		IF bSetupModeA THEN
			CASE nSetupModeAStep OF
			0:	(*MM_SetupModeA *)
				IF bMachineFault THEN
					(* Doors closed handled in Faults *)
					bSetupA:=FALSE;
					bACoolantSolenoid := FALSE;
					bSetupModeA:=FALSE;
					nManualModeState:=MM_Nothing;
				(* High Pressure Pump must be running *)
				ELSIF NOT bHighPressureMotorRunning THEN
					bSetupA:=FALSE;
					bACoolantSolenoid := FALSE;
					nManualModeState:=MM_Nothing;
					bSetupModeA:=FALSE;
					nModeError := Er_CoolantOff;
				(* Parts Must be Present *)
				ELSIF NOT(nAEjectorRetractedState=0) OR NOT(nAEjectorAdvancedState=7)
				THEN
					bSetupA:=FALSE;
					bACoolantSolenoid := FALSE;
					nManualModeState:=MM_Nothing;
					bSetupModeA:=FALSE;
					nModeError := Er_SetupError;
					nSetupErrorID:=1;
				(* Parts Must be Clamped *)
				ELSIF NOT(bPS617) THEN
					bSetupA:=FALSE;
					bACoolantSolenoid := FALSE;
					nManualModeState:=MM_Nothing;
					bSetupModeA:=FALSE;
					nModeError := Er_SetupError;
					nSetupErrorID:=2;
				(* UnClamp PS Must be Off *)
				ELSIF bPS616 THEN
					bSetupA:=FALSE;
					bACoolantSolenoid := FALSE;
					nManualModeState:=MM_Nothing;
					bSetupModeA:=FALSE;
					nModeError := Er_SetupError;
					nSetupErrorID:=3;
				(* Exit When Drill Return is Pressed *)
				ELSIF NOT(bPB4ADrillReturn) OR NOT(bPB4BDrillReturn) THEN
					bACoolantSolenoid := FALSE;
					bSetupA:=FALSE;
					bSetupModeA:=FALSE;
					nManualModeState:=MM_Nothing;
				(* If PB is pressed again then move to MMSetup with Spindle *)
				ELSIF fbSetupModeATimer.Q AND bEnterSetupPB_A THEN
					nSetupModeAStep:=1;
					bVFD_ARun:=TRUE;
				(* Turn on the In Setup bit and the solenoid *)
				ELSE
					bACoolantSolenoid := TRUE;
					bSetupA:=TRUE;
				END_IF

			1:	(*	MM_SetupModeAWSpindle		*)
				nVFDControlRPM:=LREAL_TO_UINT(fRPMRequest);
				(* The Setup can be canceled by Drill Retrun of Fault Reset *)
				IF bMachineFault OR NOT(bPB4ADrillReturn) OR NOT(bPB4BDrillReturn) OR bFaultResetPB THEN
					bACoolantSolenoid :=FALSE;
					bVFD_ARun:=FALSE;
					bSetupA:=FALSE;
					bSetupModeA:=FALSE;
					nSetupModeAStep:=0;
					nManualModeState:=MM_Nothing;
				END_IF
			END_CASE	(* nSetupModeAStep *)
		END_IF (*bSetupmodeA *)

		(* MM_SetupModeB*)
		IF bSetupModeB THEN
			CASE nSetupModeBStep OF
			0:	(*MM_SetupModeB *)
				IF bMachineFault THEN
					(* Doors closed handled in Faults *)
					bSetupB:=FALSE;
					bBCoolantSolenoid := FALSE;
					bSetupModeB:=FALSE;
					nManualModeState:=MM_Nothing;
				(* High Pressure Pump must be running *)
				ELSIF NOT bHighPressureMotorRunning THEN
					bSetupB:=FALSE;
					bBCoolantSolenoid := FALSE;
					nManualModeState:=MM_Nothing;
					bSetupModeB:=FALSE;
					nModeError := Er_CoolantOff;
				(* Parts Must be Present *)
				ELSIF NOT(nBEjectorRetractedState=0) OR NOT(nBEjectorAdvancedState=7)
				THEN
					bSetupB:=FALSE;
					bBCoolantSolenoid := FALSE;
					nManualModeState:=MM_Nothing;
					bSetupModeB:=FALSE;
					nModeError := Er_SetupError;
					nSetupErrorID:=1;
				(* Parts Must be Clamped *)
				ELSIF NOT(bPS727) THEN
					bSetupB:=FALSE;
					bBCoolantSolenoid := FALSE;
					nManualModeState:=MM_Nothing;
					bSetupModeB:=FALSE;
					nModeError := Er_SetupError;
					nSetupErrorID:=2;
				(* Unclamped PS Off*)
				ELSIF bPS726 THEN
					bSetupB:=FALSE;
					bBCoolantSolenoid := FALSE;
					nManualModeState:=MM_Nothing;
					bSetupModeB:=FALSE;
					nModeError := Er_SetupError;
					nSetupErrorID:=3;
				(* Exit When Drill Return is Pressed *)
				ELSIF NOT(bPB4ADrillReturn) OR NOT(bPB4BDrillReturn) THEN
					bBCoolantSolenoid := FALSE;
					bSetupB:=FALSE;
					bSetupModeB:=FALSE;
					nManualModeState:=MM_Nothing;
				(* If PB is pressed again then move to MMSetup with Spindle *)
				ELSIF fbSetupModeBTimer.Q AND bEnterSetupPB_B THEN
					nSetupModeBStep:=1;
					bVFD_BRun:=TRUE;
				(* Turn on the In Setup bit and the solenoid *)
				ELSE
					bBCoolantSolenoid := TRUE;
					bSetupB:=TRUE;
				END_IF

			1:	(*MM_SetupModeBWSpindle*)
				nVFDControlRPM:=LREAL_TO_UINT(fRPMRequest);
				(* The Setup can be canceled by Drill Retrun of Fault Reset *)
				IF bMachineFault OR NOT(bPB4ADrillReturn) OR NOT(bPB4BDrillReturn) OR bFaultResetPB THEN
					bBCoolantSolenoid :=FALSE;
					bVFD_BRun:=FALSE;
					bSetupB:=FALSE;
					bSetupModeB:=FALSE;
					nSetupModeBStep:=0;
					nManualModeState:=MM_Nothing;
				END_IF
			END_CASE	(* nSetupModeAStep *)
		END_IF (*bSetupmodeB *)

		MM_SetZAZero:
			IF bMachineFault THEN
				bZAAxisSetZero := FALSE;
				nManualModeState:=MM_Nothing;
			ELSIF fbZAAxisSetZero.Error THEN
				nModeError := Er_ZAHomeError;
				bZAAxisSetZero := FALSE;
				nManualModeState:=MM_Nothing;
			ELSIF fbZAAxisSetZero.Done THEN
				bZAAxisSetZero := FALSE;
				nManualModeState:=MM_Nothing;
			ELSE
				bZAAxisSetZero := TRUE;
			END_IF

		MM_SetZBZero:
			IF bMachineFault THEN
				bZBAxisSetZero := FALSE;
				nManualModeState:=MM_Nothing;
			ELSIF fbZBAxisSetZero.Error THEN
				nModeError := Er_ZBHomeError;
				bZBAxisSetZero := FALSE;
				nManualModeState:=MM_Nothing;
			ELSIF fbZBAxisSetZero.Done THEN
				bZBAxisSetZero := FALSE;
				nManualModeState:=MM_Nothing;
			ELSE
				bZBAxisSetZero := TRUE;
			END_IF

		MM_MoveZAToZero:
			IF bMachineFault THEN
				bZAAxisMove := FALSE;
				nManualModeState:=MM_Nothing;
			ELSIF fbZAAxisMove.Error THEN
				nModeError := Er_ZAMoveError;
				bZAAxisMove := FALSE;
				nManualModeState:=MM_Nothing;
			ELSIF fbZAAxisMove.Done THEN
				bZAAxisMove := FALSE;
				nManualModeState:=MM_Nothing;
			ELSE
				bZAAxisMove := TRUE;
				fZAMovePosition := 0.0;
				fZAMoveVelocity := 25.0;
			END_IF

		MM_MoveZBToZero:
			IF bMachineFault THEN
				bZBAxisMove := FALSE;
				nManualModeState:=MM_Nothing;
			ELSIF fbZBAxisMove.Error THEN
				nModeError := Er_ZBMoveError;
				bZBAxisMove := FALSE;
				nManualModeState:=MM_Nothing;
			ELSIF fbZBAxisMove.Done THEN
				bZBAxisMove := FALSE;
				nManualModeState:=MM_Nothing;
			ELSE
				bZBAxisMove := TRUE;
				fZBMovePosition := 0.0;
				fZBMoveVelocity := 25.0;
			END_IF

		MM_CoolantOn:
			(* Make sure the Clean tank level has been on for 2 seconds so that we
				don't draw the level down to quickly when we start the High Pressure Pump *)
			fbCleanTankLevelDelay(IN:=bCleanTankLevel, PT:=t#2s);
			(* If the Coolant Stop PB is pressed while in startup *)
			IF bCoolantStopPB THEN
				nManualModeState:=MM_CoolantOff;
			END_IF

			IF bMachineFault THEN
				bHPCoolantStart_A :=FALSE;
				bHPCoolantStart_B :=FALSE;
				bTransferPumpMotorControl:=FALSE;
				bHighPressureMotorControl:=FALSE;
				nManualModeState:=MM_Nothing;
			(* S1: Start the transfer pump and Turn on the Soft Start Solenoid Valves *)
			ELSIF NOT(fbSoftStartTimer.Q) AND NOT(fbSoftStartTimer2.Q) THEN
				bHPCoolantStart_A :=TRUE;
				bHPCoolantStart_B :=TRUE;
				bTransferPumpMotorControl:=TRUE;
			(* S2: After 5 seconds turn on high pressure Motor *)
			(* Note: We can stay here until we get a fault such as Low Tank Level *)
			ELSIF fbSoftStartTimer.Q AND NOT(fbSoftStartTimer2.Q) AND fbCleanTankLevelDelay.Q
				AND NOT(bCoolantTempWarning) AND bCoolantTankOverflow
			THEN
				bHighPressureMotorControl:=TRUE;
			(* S3: After 5 more seconds Turn off the Soft Start Solenoids *)
			ELSIF fbSoftStartTimer2.Q THEN
				bHPCoolantStart_A :=FALSE;
				bHPCoolantStart_B :=FALSE;
				bChipConveyorMotorControl:=TRUE;
				nManualModeState:=MM_Nothing;
			END_IF

		MM_CoolantOff:
			(*	Turn off High Pressure Motor *)
			bHighPressureMotorControl:=FALSE;
			(* Do not shut off the transfer pump until the coolant temp is below the warning *)
			IF bCoolantTempWarning OR bCoolantTempFault THEN
				bChipConveyorMotorControl:=FALSE;
				nManualModeState:=MM_Nothing;
			ELSIF NOT(bHighPressureMotorOn) THEN
				(*	Turn off Transfer Pump *)
				bTransferPumpMotorControl:=FALSE;
				(*	Done *)
				IF NOT(bTransferPumpOn) THEN
					bChipConveyorMotorControl:=FALSE;
					nManualModeState:=MM_Nothing;
				END_IF
			END_IF

		MM_HomeAutomation:
			IF bMachineFault THEN
				nHomeAutomationStep:=0;
				bWAAxisHome:=FALSE;
				bWBAxisHome:=FALSE;
				bUAxisHome:=FALSE;
				(* Trigger MCStop of Axis.  The bits are turned false when done in respective control *)
				bWAStop:=TRUE;
				bWAStop:=TRUE;
				bUStop:=TRUE;
			ELSE
				CASE nHomeAutomationStep OF
				0: (* Trigger Home of WA and WB Axis *)
					IF bSideAEnabled THEN
						bWAAxisHome:=TRUE;	(* Turned off in P_Tailstock Control PRG *)
					END_IF
					IF bSideBEnabled THEN
						bWBAxisHome:=TRUE;	(* Turned off in P_Tailstock Control PRG *)
					END_IF
					nHomeAutomationStep:=nHomeAutomationStep+1;
	
				1: (* After 1 second then start Homing the U Axis, This assures enough clearance *)
					fbHomeTimer(IN:=TRUE, PT:=t#2s);
					IF fbHomeTimer.Q THEN
						fbHomeTimer(IN:=FALSE);
						(* If an error occurs in either of the Axis we want leave the homing operation *)
						IF fbWAAxisHome.Error OR fbHomeWB.Error THEN
							nHomeAutomationStep:=0;
							nManualModeState:=MM_Nothing;
						(* No Errors Move On *)
						ELSE
							bUAxisHome:=TRUE;
							nHomeAutomationStep:=nHomeAutomationStep+1;
						END_IF
					END_IF
	
				2: (* Check for Done bits of the three Axis *)
					fbHomeTimer(IN:=TRUE, PT:=t#90s);
					(* When All Axis are Homed we return *)
					IF (stWAAxis.NcToPlc.StateDWord.1 AND stWBAxis.NcToPlc.StateDWord.1 AND stUAxis.NcToPlc.StateDWord.1) OR
						(* or if an Error occurs *)
						 fbWAAxisHome.Error OR fbHomeWB.Error OR fbTransferAxisHome.Error OR
						(* or if Homing takes too long *)
						fbHomeTimer.Q
					THEN
						fbHomeTimer(IN:=FALSE);
						nHomeAutomationStep:=0;
						nManualModeState:=MM_Nothing;
						IF fbHomeTimer.Q THEN
							nModeError:=Er_HomeTimeout;
						END_IF
					END_IF

				END_CASE	(* nHomeAutomationStep *)
			END_IF	(* Fault check of MM_HomeAutomation *)

		END_CASE	(* Manual Mode State *)

	(*********		AUTOMATIC MODE 		***********)
	ELSE
		CASE nAutoModeState OF
		AM_NotInCycle:
			(* If we have a fault we Exit Auto Mode *)
			IF bMachineFault THEN
				bMachineMode:=FALSE;
			(* We disable cycle start when we have warings *)
			ELSIF bCycleStartControlEnable AND NOT(bMachineWarning)  THEN
				(* Doors will fault if not closed in cycle *)
				nAutoModeState:=AM_RetractZAxis;
			END_IF

		AM_RetractZAxis:
			IF bMachineFault THEN
				bZAAxisMove:= FALSE;
				bZBAxisMove:= FALSE;
				bZAStop := TRUE;
				bZBStop := TRUE;
				nAutoModeState:=AM_NotInCycle;
			ELSE
				(* Move Z axis to Drill Tip Offset Position *)
				IF bSideAEnabled THEN
					bZAAxisMove:= TRUE;
					fZAMovePosition := fDrillTipOffset;
					fZAMoveVelocity := 25;
				END_IF
				IF bSideBEnabled THEN
					bZBAxisMove:= TRUE;
					fZBMovePosition := fDrillTipOffset;
					fZBMoveVelocity := 25;
				END_IF
				(* Stop Axis and Fault if Move Error *)
				IF (bSideAEnabled AND fbZAAxisMove.Error) THEN
					bZAAxisMove:= FALSE;
					nModeError := Er_ZAHomeError;
					bZAStop:=TRUE;	(* Issue a Stop Axis *)
					bZBAxisMove:= FALSE;
					bMachineMode:=FALSE;	(* Go to Manual Mode *)
				ELSIF (bSideBEnabled AND fbZBAxisMove.Error) THEN
					bZBAxisMove:= FALSE;
					nModeError := Er_ZAHomeError;
					bZBStop:=TRUE;	(* Issue a Stop Axis *)
					bZAAxisMove:= FALSE;
					bMachineMode:=FALSE;	(* Go to Manual Mode *)
				(* If Move Done we Go Into Cycle *)
				ELSIF (NOT(bSideAEnabled) OR fbZAAxisMove.Done) AND
					(NOT(bSideBEnabled) OR fbZBAxisMove.Done) THEN
					bZAAxisMove:= FALSE;
					bZBAxisMove:= FALSE;
					nAutoModeState:=AM_InCycle;
				END_IF
			END_IF

		AM_InCycle:
			(* These Things Happen While In Cycle *)
			fbCoolantTimer(IN:=bCoolantTimer , PT:=tCoolantTime);
			fbCycleTimer(IN:=bCycleTimer , PT:=t#10h);
			(* If the Load confirm PB has been pressed and the parts are there,  then Set a bit for Load Confirm *)
			IF ( sLoadSideSet = 'A' AND bPB1AConfirm AND
				(NOT(bSideAEnabled) OR bProx410 AND bProx411 AND bProx412) AND
				(NOT(bSideBEnabled) OR bProx413 AND bProx414 AND bProx415) ) OR
				(sLoadSideSet ='B' AND bPB1BConfirm AND
				( NOT(bSideAEnabled) OR bProx510 AND bProx511 AND bProx512) AND
				(NOT(bSideBEnabled) OR bProx513 AND bProx514 AND bProx515) )
			THEN
				bLoadPartsConfirmed:= TRUE;	(* Turned Off in Transfer Control *)
			(* Else Set a Warning that Parts are Missing when the PB pressed
				We want to ignore the PB if we have already confirmed parts loaded *)
			ELSIF NOT bLoadPartsConfirmed AND
				( sLoadSideSet = 'A' AND fbPB1AConfirmRTrig.Q) OR
				(sLoadSideSet ='B' AND fbPB1BConfirmRTrig.Q)
			THEN
				nModeError:=Er_LoadPartMissing;
			END_IF
			(* If the Unloadoad confirm PB's have been pressed and there are no parts,  then Set a bit for Unload Confirm *)
			IF (sLoadSideSet = 'B' AND fbPB1AConfirmRTrig.Q AND
				NOT(bProx410 OR bProx411 OR bProx412 OR bProx413 OR bProx414 OR bProx415) ) OR
				(sLoadSideSet ='A' AND fbPB1BConfirmRTrig.Q AND
				NOT(bProx510 OR bProx511 OR bProx512 OR bProx513 OR bProx514 OR bProx515) )
			THEN
				bUnloadPartsConfirmed:= TRUE;
			(* Else set a Warning that Parts are present *)
			ELSIF (sLoadSideSet = 'B' AND fbPB1AConfirmRTrig.Q) OR (sLoadSideSet ='A' AND fbPB1BConfirmRTrig.Q) THEN
				nModeError:=Er_UnloadPartPresent;
			END_IF

			(*	Implement Auto Cycle Stuff Here *)
			CASE nAutoCycleStep OF
			AC_Init:
				bCycleStartControlHold:=FALSE;
				bCycleStartControlReset:=FALSE;
				bCycleTimer:=FALSE;
				(* Check Faults *)
				IF bMachineFault THEN (* Added V1.5 *)
					bInCycle:=FALSE;
					bMachineMode:=FALSE;
					bCycleStartControlReset:=TRUE;
					nAutoModeState:=AM_NotInCycle;
				ELSIF bLoadPartsConfirmed THEN
					nDrillStep := 0;
					bInCycle:=TRUE;
					nAutoCycleStep:=AC_TransferParts;
				END_IF

			AC_TransferParts:
				(* When Cycle Counter Reached and not Cell Runout we Fault *)
				IF (nCyclesComplete >= nMaxCycles) AND NOT bCellRunoutRequest THEN
					nModeError:= Er_MaxCyclesReached;
					nAutoCycleStep:=AC_Init;
					nAutoModeState:=AM_NotInCycle;
					bMachineMode:=FALSE;
					bCycleStartControlReset:=TRUE;
					bCycleStartControlHold:=FALSE;
					bCycleWatchdogTimer := FALSE;
					bInCycle:=FALSE;
					bCycleTimer:=FALSE;
					bDisplayUnloadConf := FALSE;
				ELSE
					bCycleTimer:=TRUE;
					IF bMachineFault OR fbCycleWatchdogTimer.Q THEN
						nAutoCycleStep:=AC_Init;
						bInCycle:=FALSE;
						bMachineMode:=FALSE;
						bCycleStartControlReset:=TRUE;
						bCycleStartControlHold:=FALSE;
						bCycleWatchdogTimer := FALSE;
						bCycleTimer:=FALSE;
						bDisplayUnloadConf := FALSE;
						bAutoTransferPartsToDrill:=FALSE;
						nAutoModeState:=AM_NotInCycle;
					(* At Unload Position and UP, So Go to Clamp *)
					ELSIF bTransferAtUnloadIndicator AND
						bProx516 AND NOT(bProx517)
					THEN
						bCycleWatchdogTimer := FALSE;
						IF nCellRunoutCounter=1 AND bCellRunoutRequest THEN
							nAutoCycleStep:=AC_CellRunoutFinish;
						ELSE
							nAutoCycleStep:=AC_Clamp;
						END_IF
					(* Trigger Transfer Move *)
					ELSIF NOT bAutoTransferPartsToDrill  AND bUnloadPartsConfirmed THEN
						bDisplayUnloadConf := FALSE;
						bAutoTransferPartsToDrill:=TRUE;
						bCycleWatchdogTimer := TRUE;
						tCycleWatchdogTime := t#120s;
					(* Display Waiting on Unload Confirm Button *)
					ELSIF NOT bUnloadPartsConfirmed THEN
						bDisplayUnloadConf := TRUE;
					END_IF
				END_IF (* Max Cycles Check *)

			AC_Clamp:
				IF bMachineFault (* OR fbCycleWatchdogTimer.Q *) THEN
					nAutoCycleStep:=AC_Init;
					bInCycle:=FALSE;
					bMachineMode:=FALSE;
					bCycleStartControlReset:=TRUE;
					bCycleStartControlHold:=FALSE;
					bCycleTimer:=FALSE;
					bCycleWatchdogTimer := FALSE;
					bAutoClampAStart:=FALSE;
					bAutoClampBStart:=FALSE;
					nAutoModeState:=AM_NotInCycle;
				(* Done Clamping so Go To Coolant On *)
				ELSIF(bAutoClampADone OR NOT(bSideAEnabled)) AND
						(bAutoClampBDone OR NOT(bSideBEnabled)) THEN
					bAutoTransferDownAndLoad := TRUE;
					bCycleWatchdogTimer := FALSE;
					nAutoCycleStep:=AC_CoolantOn;
				(* Trigger Clamping *)
				ELSE
					bCycleWatchdogTimer := TRUE;
					tCycleWatchdogTime := t#30s;
					IF bSideAEnabled THEN
						bAutoClampAStart:=TRUE;
					END_IF
					IF bSideBEnabled THEN
						bAutoClampBStart:=TRUE;
					END_IF
				END_IF

			AC_CoolantOn:
				IF bMachineFault OR fbCycleWatchdogTimer.Q THEN
					nAutoCycleStep:=AC_Init;
					bInCycle:=FALSE;
					bMachineMode:=FALSE;
					bCycleStartControlReset:=TRUE;
					bCycleStartControlHold:=FALSE;
					bCycleTimer:=FALSE;
					bCycleWatchdogTimer := FALSE;
					bAutoClampAStart:=FALSE;
					bAutoClampBStart:=FALSE;
					bACoolantSolenoid:=FALSE;
					bBCoolantSolenoid:=FALSE;
					bAutoTransferDownAndLoad := FALSE;
					IF fbCycleWatchdogTimer.Q THEN
						nModeError:=Er_AMCoolantTimeout;
					END_IF
					nAutoModeState:=AM_NotInCycle;
				(* S2: When Pressure Switch On Delay then Turn Spindles On *)
				ELSIF (fbPS1DelayTON.Q OR NOT(bSideAEnabled)) AND
						(fbPS2DelayTON.Q OR NOT(bSideBEnabled)) THEN
					bCycleWatchdogTimer := FALSE;
					nAutoCycleStep:=AC_SpindleOn;
				(* S1: Turn on the Coolant and start the watchdog Timer
					Set the PS delay timer *)
				ELSE
					IF bSideAEnabled THEN
						bACoolantSolenoid:=TRUE;
					END_IF
					IF bSideBEnabled THEN
						bBCoolantSolenoid:=TRUE;
					END_IF
					tCoolantTime:= t#1.5s;
					bCycleWatchdogTimer := TRUE;
					tCycleWatchdogTime := t#15s;
				END_IF

			AC_SpindleOn:
				nVFDControlRPM:=LREAL_TO_UINT(fRPMRequest);
				IF bMachineFault OR fbCycleWatchdogTimer.Q THEN
					nAutoCycleStep:=AC_Init;
					bInCycle:=FALSE;
					bMachineMode:=FALSE;
					bCycleStartControlReset:=TRUE;
					bCycleStartControlHold:=FALSE;
					bCycleTimer:=FALSE;
					bCycleWatchdogTimer := FALSE;
					bAutoClampAStart:=FALSE;
					bAutoClampBStart:=FALSE;
					bACoolantSolenoid:=FALSE;
					bBCoolantSolenoid:=FALSE;
					bVFD_ARun:=FALSE;
					bVFD_BRun:=FALSE;
					bAutoTransferDownAndLoad := FALSE;
					IF fbCycleWatchdogTimer.Q THEN
						nModeError:=Er_VFDUpToSpeedTimeout;
					END_IF
					nAutoModeState:=AM_NotInCycle;
				(* S2: Once up to Speed then Drill *)
				ELSIF (fbUpToSpeedATON.Q OR NOT(bSideAEnabled)) AND
						(fbUpToSpeedBTON.Q OR NOT(bSideBEnabled)) THEN
					bCycleWatchdogTimer := FALSE;
					nAutoCycleStep:=AC_Drill;
				(* S1: Turn on Spindles *)
				ELSE
					IF bSideAEnabled THEN
						bVFD_ARun := TRUE;
					END_IF
					IF bSideBEnabled THEN
						bVFD_BRun := TRUE;
					END_IF
					tCycleDelayTime := t#250ms;
				END_IF

			AC_Drill:
				(* Safety interlock: while drilling, keep transfer commands disabled so the part cannot move with drills engaged. *)
				bAutoTransferPartsToDrill:=FALSE;
				bAutoTransferDownAndLoad:=FALSE;
				IF bMachineFault  AND
					(*Faults Array 4 are ones that should not stop the drill cycle *)
					NOT( nActiveFaults[4]>0
						AND nActiveFaults[1]=0
						AND nActiveFaults[2]=0
						AND nActiveFaults[3]=0)
				THEN
					nAutoCycleStep:=AC_DrillReturn;
					nDrillStep := 0;
					bInCycle:=FALSE;
					bCycleStartControlReset:=TRUE;
					bCycleStartControlHold:=FALSE;
					bCycleTimer:=FALSE;
					bCycleWatchdogTimer := FALSE;
					bAutoClampAStart:=FALSE;
					bAutoClampBStart:=FALSE;
					bACoolantSolenoid:=FALSE;
					bBCoolantSolenoid:=FALSE;
					bZAAxisMove:=FALSE;
					bZBAxisMove:=FALSE;
					bZAStop := TRUE;
					bZBStop := TRUE;
					bVFD_ARun:=FALSE;
					bVFD_BRun:=FALSE;
					bDwellTime:= FALSE;
					bAutoTransferDownAndLoad := FALSE;
				ELSE
					(* S1: Move to Strart Depth at Startfeed *)
					(* S2: Wait for Move Done bit *)
					(* S3: Move to Finish Depth at Finish Feed *)
					(* S4: Wait for Move Done bit *)
					(* S5: If Dead Spindle Retract Then-Turn off Spindles *)
					(* T5: VFD's at Zero Speed *)
					(* S6: If Not Dead Spindle Retract then use Dwell Timer *)
					CASE nDrillStep OF
					0: (* S1: Set Execute for Z Axis *)
						IF bSideAEnabled THEN
							bZAAxisMove:=TRUE;
							fZAMovePosition:= fStartDepth;
							fZAMoveVelocity:= fStartFeed/60;
						END_IF
						IF bSideBEnabled THEN
							bZBAxisMove:=TRUE;
							fZBMovePosition:= fStartDepth;
							fZBMoveVelocity:= fStartFeed/60;
						END_IF
						(* T1: Wait for Busy bit *)
						IF (fbZAAxisMove.Busy OR NOT(bSideAEnabled)) AND
							(fbZBAxisMove.Busy OR NOT(bSideBEnabled)) THEN
							nDrillStep:=nDrillStep+1;
						END_IF

					1:(* S2: Wait for Move Start Depth Done bit *)
						IF (fbZAAxisMove.Done OR NOT(bSideAEnabled)) AND
							(fbZBAxisMove.Done OR NOT(bSideBEnabled)) THEN
							bZAAxisMove:=FALSE;
							bZBAxisMove:=FALSE;
							nDrillStep:=nDrillStep+1;
						END_IF

					2: (* S3: Move to Finish Depth at Finish Feed *)
						IF bSideAEnabled THEN
							bZAAxisMove:=TRUE;
							fZAMovePosition:= fFinishDepth;
							fZAMoveVelocity:= fFinishFeed/60;
						END_IF
						IF bSideBEnabled THEN
							bZBAxisMove:=TRUE;
							fZBMovePosition:= fFinishDepth;
							fZBMoveVelocity:= fFinishFeed/60;
						END_IF
						(* T1: Wait for Busy bit *)
						IF (fbZAAxisMove.Busy OR NOT(bSideAEnabled)) AND
							(fbZBAxisMove.Busy OR NOT(bSideBEnabled)) THEN
							nDrillStep:=nDrillStep+1;
						END_IF

					3: (* S4: Wait for Move Done bit *)
						IF (fbZAAxisMove.Done OR NOT(bSideAEnabled)) AND
							(fbZBAxisMove.Done OR NOT(bSideBEnabled)) THEN
							bZAAxisMove:=FALSE;
							bZBAxisMove:=FALSE;
							nDrillStep:=nDrillStep+1;
						END_IF

					4: (* If Dead Spindle Retract then go to Step 5, Else Step 6 *)
						IF bSpindleRetractMode THEN
							nDrillStep:=nDrillStep+1;
						ELSE
							nDrillStep:=6;
						END_IF

					5: (* S5: Turn off Spindles *)
						(* Turn off the VFD Run singnals *)
						bVFD_ARun:=FALSE;
						bVFD_BRun:=FALSE;
						tCycleWatchdogTime := t#5s;
						bCycleWatchdogTimer:=TRUE;
						IF (NOT(bSideAEnabled) OR (stVFD_A1DriveInfo.nActualSpeed < 5) OR
							(stVFD_A2DriveInfo.nActualSpeed < 5) OR (stVFD_A3DriveInfo.nActualSpeed < 5) )
							AND (NOT(bSideBEnabled) OR  (stVFD_A1DriveInfo.nActualSpeed < 5) OR
							(stVFD_A2DriveInfo.nActualSpeed < 5) OR (stVFD_A3DriveInfo.nActualSpeed < 5) )
						THEN
							bCycleWatchdogTimer := FALSE;
							nDrillStep:=0;
							nAutoCycleStep:=AC_Retract;
						(* If This took too long then jump to next step *)
						ELSIF fbCycleWatchdogTimer.Q THEN
							bCycleWatchdogTimer := FALSE;
							nDrillStep:=0;
							nAutoCycleStep:=AC_Retract;
						END_IF

					6: (* S6: Dwell Timer *)
						IF fDwellTime > 0.0 THEN
							bDwellTime:= TRUE;
							fbDwellTimeTON(IN:=bDwellTime, PT:=LREAL_TO_TIME(fDwellTime) );
							IF fbDwellTimeTON.Q THEN
								bDwellTime:= FALSE;
								nDrillStep:=0;
								nAutoCycleStep:=AC_Retract;
							END_IF
						ELSE (* No Dwell Time *)
							nDrillStep:=0;
							nAutoCycleStep:=AC_Retract;
						END_IF

					END_CASE
				END_IF

			AC_DrillReturn:
				(* Keep transfer disabled until Z axes have returned to drill tip offset. *)
				bAutoTransferPartsToDrill:=FALSE;
				bAutoTransferDownAndLoad:=FALSE;
				CASE nDrillReturnCount OF
				0: (* Wait for the Stop to finish and Move to Drill Tip Offset *)
					IF NOT bZAStop AND NOT bZBStop THEN
						bZAAxisMove:=TRUE;
						bZBAxisMove:=TRUE;
						fZAMovePosition:=fDrillTipOffset;
						fZBMovePosition:=fDrillTipOffset;
						fZAMoveVelocity:=50;
						fZBMoveVelocity:=50;
						nDrillReturnCount:=nDrillReturnCount+1;
					END_IF

				1: (* Wait for move to be done *)
					IF fbZAAxisMove.Done AND fbZBAxisMove.Done THEN
						bZAAxisMove:=FALSE;
						bZBAxisMove:=FALSE;
						bMachineMode:=FALSE;
						nAutoModeState:=AM_NotInCycle;
						nDrillReturnCount:=0;
					END_IF
				END_CASE


			AC_Retract:
				(* Keep transfer disabled until drills are fully retracted and spindle/coolant shutdown is complete. *)
				bAutoTransferPartsToDrill:=FALSE;
				bAutoTransferDownAndLoad:=FALSE;
				IF bMachineFault  AND
					(*Faults Array 4 are ones that should not stop the drill cycle *)
					NOT( (nActiveFaults[4]>0)
						AND nActiveFaults[1]=0
						AND nActiveFaults[2]=0
						AND nActiveFaults[3]=0)
				THEN
					nAutoCycleStep:=AC_Init;
					nDrillStep := 0;
					bInCycle:=FALSE;
					bMachineMode:=FALSE;
					bCycleStartControlReset:=TRUE;
					bCycleStartControlHold:=FALSE;
					bCycleTimer:=FALSE;
					bCycleWatchdogTimer := FALSE;
					bAutoClampAStart:=FALSE;
					bAutoClampBStart:=FALSE;
					bACoolantSolenoid:=FALSE;
					bBCoolantSolenoid:=FALSE;
					bZAAxisMove:=FALSE;
					bZBAxisMove:=FALSE;
					bZAStop := TRUE;
					bZBStop := TRUE;
					bVFD_ARun:=FALSE;
					bVFD_BRun:=FALSE;
					bAutoTransferDownAndLoad := FALSE;
					nAutoModeState:=AM_NotInCycle;
				(* T1: Move Done Bit *)
				ELSIF (fbZAAxisMove.Done OR NOT(bSideAEnabled)) AND
						(fbZBAxisMove.Done OR NOT(bSideBEnabled)) THEN
					bZAAxisMove:=FALSE;
					bZBAxisMove:=FALSE;
					nAutoCycleStep:=AC_SpindleOff;
				(* S1: Move to Start Position *)
				ELSE
					IF bSideAEnabled THEN
						bZAAxisMove:=TRUE;
						fZAMovePosition:= (0.0 + fDrillTipOffset);
						fZAMoveVelocity:= fRetractRate/60;
					END_IF
					IF bSideBEnabled THEN
						bZBAxisMove:=TRUE;
						fZBMovePosition:= (0.0 + fDrillTipOffset);
						fZBMoveVelocity:= fRetractRate/60;
					END_IF
				END_IF

			AC_SpindleOff:
				(* Turn off the VFD Run singnals *)
				bVFD_ARun:=FALSE;
				bVFD_BRun:=FALSE;
				nAutoCycleStep:=AC_CoolantOff;

			AC_CoolantOff:
				(* Turn off the Coolant Valves *)
				bACoolantSolenoid:=FALSE;
				bBCoolantSolenoid:=FALSE;
				(* Add a time delay so we don't squirt coolant before Unclamping *)
				bCoolantTimer:=TRUE;
				tCoolantTime:=t#250ms;
				IF ( bMachineFault  AND
					(*Faults Array 4 are ones that should not stop the drill cycle *)
					NOT( (nActiveFaults[4]>0)
						AND nActiveFaults[1]=0
						AND nActiveFaults[2]=0
						AND nActiveFaults[3]=0) )
					OR fbCycleWatchdogTimer.Q
				THEN
					nAutoCycleStep:=AC_Init;
					bInCycle:=FALSE;
					bMachineMode:=FALSE;
					bCoolantTimer:=FALSE;
					bCycleStartControlReset:=TRUE;
					bCycleStartControlHold:=FALSE;
					bCycleTimer:=FALSE;
					bCycleWatchdogTimer := FALSE;
					bAutoClampAStart:=FALSE;
					bAutoClampBStart:=FALSE;
					bAutoTransferDownAndLoad := FALSE;
					IF fbCycleWatchdogTimer.Q THEN
						nModeError:=Er_MMCoolantValveStopTimeout;
					END_IF
					nAutoModeState:=AM_NotInCycle;
				ELSIF NOT(bACoolantPressure) AND NOT(bBCoolantPressure) THEN
					bCycleWatchdogTimer := FALSE;
					bCoolantTimer:=FALSE;
					nCyclesComplete:=nCyclesComplete+1;
					IF bSideAEnabled THEN
						nPartsCompleteTotal:=nPartsCompleteTotal+3;
						nPartsCompleteA1:=nPartsCompleteA1+1;
						nPartsCompleteA2:=nPartsCompleteA2+1;
						nPartsCompleteA3:=nPartsCompleteA3+1;
					END_IF
					IF bSideBEnabled THEN
						nPartsCompleteTotal:=nPartsCompleteTotal+3;
						nPartsCompleteB1:=nPartsCompleteB1+1;
						nPartsCompleteB2:=nPartsCompleteB2+1;
						nPartsCompleteB3:=nPartsCompleteB3+1;
					END_IF
					nAutoCycleStep:=AC_Unclamp;
				ELSE
					bCycleWatchdogTimer := TRUE;
					tCycleWatchdogTime := t#10s;
				END_IF

			AC_Unclamp:
				(* Turn off the Clamp Starts *)
				bAutoClampAStart:=FALSE;
				bAutoClampBStart:=FALSE;
				IF ( bMachineFault  AND
					(*Faults Array 4 are ones that should not stop the drill cycle *)
					NOT( (nActiveFaults[4]>0)
						AND nActiveFaults[1]=0
						AND nActiveFaults[2]=0
						AND nActiveFaults[3]=0) )
					OR fbCycleWatchdogTimer.Q
				THEN
					nAutoCycleStep:=AC_Init;
					bInCycle:=FALSE;
					bMachineMode:=FALSE;
					bCycleStartControlReset:=TRUE;
					bCycleStartControlHold:=FALSE;
					bCycleTimer:=FALSE;
					bCycleWatchdogTimer := FALSE;
					bAutoTransferDownAndLoad := FALSE;
					bAutoUpDelayWhileUnclamp := FALSE;
					bAutoUnclampAStart:=FALSE;
					bAutoUnclampBStart:=FALSE;
					nAC_UnclampStep:=0;
					IF fbCycleWatchdogTimer.Q THEN
						nModeError:=Er_AMUnclampTimeout;
					END_IF
					nAutoModeState:=AM_NotInCycle;
				END_IF

				CASE nAC_UnclampStep OF
				0: (* Wait for Transfer to beAt Load Station and Up *)
					IF bTransferAtLoadIndicator AND
						fbProx516TON.Q AND NOT(bProx517)
					THEN
						nAC_UnclampStep := nAC_UnclampStep + 1;
					END_IF

				1: (* Once Delay timer done we can start the Unclamp process *)
					(* Watchdog happens in FB, so we need to make this one longer -
						not necessary, but did not want to remove without parts to run. *)
					bCycleWatchdogTimer := TRUE;
					tCycleWatchdogTime := t#15s;
					(* Unclamp the sides that are enabled *)
					IF bSideAEnabled THEN
						bAutoUnclampAStart:=TRUE;
					END_IF
					IF bSideBEnabled THEN
						bAutoUnclampBStart:=TRUE;
					END_IF
					bUnclampDelayTimer := FALSE;
					nAC_UnclampStep := nAC_UnclampStep + 1;

				2: (* Wait for Unload to be done on the sides that are enabled *)
					(* Unclamp Done, Trigger Transfer *)
					IF (NOT(bSideAEnabled) OR bAutoUnclampADone) AND
							(NOT(bSideBEnabled) OR bAutoUnclampBDone) THEN
						bAutoUnclampAStart:=FALSE;
						bAutoUnclampBStart:=FALSE;
						bCycleWatchdogTimer := FALSE;
						bAutoTransferDownAndLoad := FALSE;
						nAC_UnclampStep := 0;
						nAutoCycleStep := AC_TransferParts;
					(* Capture and Report Cycle Time *)
						tLastCycleTime:=fbCycleTimer.ET;
						nCycleTimeMinutes:=TRUNC(TIME_TO_LREAL(tLastCycleTime)/60000);
						nCycleTimeSeconds:=
							TRUNC((TIME_TO_LREAL(tLastCycleTime)-(nCycleTimeMinutes*60000))/1000);
						bCycleTimer:=FALSE;
					(* At this point if we made it trough a cycle without faults we know there are drilled parts on the side
					that are enabled.  Set a bit to track the parts to make sure they ended up at the unload station *)
						IF bSideAEnabled THEN
							bSideADrilledParts:=TRUE;
						END_IF
						IF bSideBEnabled THEN
							bSideBDrilledParts:=TRUE;
						END_IF
					END_IF

				END_CASE (* nAC_UnClampStep *)

			AC_CellRunoutFinish:
				(* If we have a machine fault at this point we want to exit Auto now *)
				IF bMachineFault THEN (* Added condition V1.5 *)
					nAutoCycleStep:=AC_Init;
					bInCycle:=FALSE;
					bMachineMode:=FALSE;
					bCycleStartControlReset:=TRUE;
					bCycleStartControlHold:=FALSE;
					bCycleTimer:=FALSE;
					bCycleWatchdogTimer := FALSE;
					bAutoTransferDownAndLoad := FALSE;
					nAutoModeState:=AM_NotInCycle;
				(* Finished so Jump out of Cycle and turn off request *)
				ELSIF bTransferAtLoadIndicator THEN
					bCellRunoutRequest:=FALSE;
					nCellRunoutCounter:= 0;
					bInCycle:=FALSE;
					nAutoCycleStep:=AC_Init;
				ELSE
					bAutoTransferDownAndLoad := TRUE;
				END_IF


			END_CASE	(* AutoCycle *)

		END_CASE	(* Auto Mode State *)

	END_IF	(*Automatic or Manual Mode*)

ELSE	(* Reset Variables from MCR Out *)
	(* Turn off Auto Mode bits *)
	bMachineMode:=FALSE;
	nAutoCycleStep:=AC_Init;
	bInCycle:=FALSE;
	bAutoTransferPartsToDrill:=FALSE;
	bAutoTransferDownAndLoad := FALSE;
	bLoadPartsConfirmed:= FALSE;
	bUnloadPartsConfirmed:= FALSE;
	bAutoClampAStart:=FALSE;
	bAutoClampBStart:=FALSE;
	bAutoUnclampAStart:=FALSE;
	bAutoUnclampBStart:=FALSE;
	nAC_UnclampStep := 0;
	nManualModeState:=MM_Nothing;
	nDrillReturnCount:=0;

	bCoolantTimer:= FALSE;
	(* Turn off Motors and Enables *)
	bVFD_A_Enable:=FALSE;
	bVFD_B_Enable:=FALSE;
	bVFD_ARun:=FALSE;
	bVFD_BRun:=FALSE;
	bHighPressureMotorControl:=FALSE;
	bTransferPumpMotorControl:=FALSE;
	bChipConveyorMotorControl:=FALSE;

	(* Turn off Solenoids *)
	bACoolantSolenoid := FALSE;
	bBCoolantSolenoid := FALSE;
	(* Turn off soft starts in case we were in Coolant Start *)
	bHPCoolantStart_A :=FALSE;
	bHPCoolantStart_B :=FALSE;

END_IF

(*	Light Tower and Fault Light Control *)
IF bMachineFault THEN
		bFaultLight:=TRUE;
		bTowerFaultLight:=TRUE;
		bTowerInCycle:=FALSE;
		bTowerNotInCycle:=FALSE;
ELSIF bMachineWarning THEN
	IF fbFaultLightBlink.ET>t#490ms THEN
		bFaultLight:=TRUE;
		bTowerFaultLight:=TRUE;
	ELSE
		bFaultLight:=FALSE;
		bTowerFaultLight:=FALSE;
	END_IF
	IF NOT(bFaultLightBlink) THEN
		bFaultLightBlink:=TRUE;
	ELSIF bFaultLightBlink AND fbFaultLightBlink.Q THEN
		bFaultLightBlink:=FALSE;
	END_IF
	bTowerInCycle:=FALSE;
	bTowerNotInCycle:=FALSE;
ELSIF bInCycle THEN
	bFaultLight:=FALSE;
	bTowerFaultLight:=FALSE;
	bTowerInCycle:=TRUE;
	bTowerNotInCycle:=FALSE;
ELSE
	bFaultLight:=FALSE;
	bTowerFaultLight:=FALSE;
	bTowerInCycle:=FALSE;
	bTowerNotInCycle:=TRUE;
END_IF
bLT2:=bTowerFaultLight;	(* Red Light on Tower *)
bLT3:=bTowerNotInCycle;	(* Amber Light on Tower *)
bLT4:=bTowerInCycle;		(* Green Light on Tower *)
bLT5:=bFaultLight;			(* Side A Panel fault light *)
bLT6:=bFaultLight;			(* Side B Panel fault light *)

(* Call Programs *)
DEMO;
P_FaultChecking;
Build_Send_Network_Data;
Build_Receive_Network_Data;
P_PartProgramStorage;
P_SaveData;
P_TransferControl;
P_TailstockControl;
P_MPGControl;

(* Call Actions *)
HydraulicPowerUnitControl;
TransferPumpMotorControl;
HighPressureMotorControl;
ChipConveyorMotorControl;
Security;
CycleStartControl;
VFDControl;
Z_AxisControl;

bSetup:=bSetupA OR bSetupB;
(* Triggers and Timers *)
fbMachineModeChangeRTrig(CLK:=bEnterAutoModePB);
fbSetupModeATimer(IN:= bSetupA , PT:=t#4s);
fbSetupModeBTimer(IN:= bSetupB , PT:=t#4s);
fbPS1DelayTON(IN:=bACoolantPressure , PT:= tCoolantTime);
fbPS2DelayTON(IN:=bBCoolantPressure , PT:= tCoolantTime);
fbUpToSpeedATON(in:=(bVFD_A1UpToSpeed AND bVFD_A2UpToSpeed AND
	 bVFD_A3UpToSpeed) , PT:=tCycleDelayTime);
fbUpToSpeedBTON(in:=(bVFD_B1UpToSpeed AND bVFD_B2UpToSpeed AND
	bVFD_B3UpToSpeed) , PT:=tCycleDelayTime);
fbSoftStartTimer(IN:= bTransferPumpMotorRunning , PT:= t#5s);
fbSoftStartTimer2(IN:= bHighPressureMotorRunning , PT:=t#5s);
fbCycleWatchdogTimer(IN:=bCycleWatchdogTimer, PT:=tCycleWatchdogTime);
fbProx517TON(IN:=bProx517, PT:=t#1.0s);			(* Delay of the Down Prox *)
fbProx516TON(IN:=bProx516, PT:=t#1.0s);			(* Delay of the Up Prox *)
fbUnclampDelayTON(IN:=bUnclampDelayTimer, PT:=t#1.0s);(* Delay the Unclamp cycle *)
fbStoppingSetupTON(IN:= bStoppingSetup, PT:=t#15s);
fbFaultLightBlink(IN:=bFaultLightBlink ,PT:=t#1000ms);
(* VFD Enable to wait for Data Valid bit, 0=Data Valid, 1= Data Invalid *)
fbVFD_ADataValid(IN:=stVFD_A1DriveInfo.bDataValid AND
					stVFD_A2DriveInfo.bDataValid AND
					stVFD_A3DriveInfo.bDataValid, PT:=t#500ms);
fbVFD_BDataValid(IN:=stVFD_B1DriveInfo.bDataValid AND
					stVFD_B2DriveInfo.bDataValid AND
					stVFD_B3DriveInfo.bDataValid, PT:=t#500ms);
(* Emerson Status Word bit 0 is Drive Healthy, *)
(* Delay of VFD starting - used to send internal reset *)
fbVFD_AHealthyTON( IN:=	stVFD_A1DriveInfo.nStatusWord.0 AND
						stVFD_A2DriveInfo.nStatusWord.0 AND
						stVFD_A3DriveInfo.nStatusWord.0,
						PT:= t#1500ms);
fbVFD_AStarting(CLK:=fbVFD_AHealthyTON.Q);
fbVFD_BHealthyTON(IN:=	stVFD_B1DriveInfo.nStatusWord.0 AND
						stVFD_B2DriveInfo.nStatusWord.0 AND
						stVFD_B3DriveInfo.nStatusWord.0,
						PT:= t#1500ms);
fbVFD_BStarting( CLK:=fbVFD_BHealthyTON.Q);
(* Trigger two Internal Fault Reset - 1) Aftre VFD's Healthy bit is true,
							2) After the VFD's have been Enabled*)
fbVFD_A_EnableTON(IN:=bVFD_A_Enable , PT:=t#1000ms);
fbVFD_B_EnableTON(IN:=bVFD_B_Enable , PT:=t#1000ms);
fbAResetInternalTrig(CLK:=fbVFD_A_EnableTON.Q);
fbBResetInternalTrig(CLK:=fbVFD_B_EnableTON.Q);
IF bSideAEnabled AND (fbVFD_AStarting.Q OR fbAResetInternalTrig.Q) THEN
	(*The bit is turned False in Fault Checking *)
	bAFaultResetInternal:=TRUE;
END_IF
(* Else side B is Enabled *)
IF bSideBEnabled AND (fbVFD_BStarting.Q OR fbBResetInternalTrig.Q) THEN
	(*The bit is turned False in Fault Checking *)
	bBFaultResetInternal:=TRUE;
END_IF

(* Rising Edge Trigger of the Load/Unload Confirm PB's *)
fbPB1AConfirmRTrig(CLK:= bPB1AConfirm);
fbPB1BConfirmRTrig(CLK:= bPB1BConfirm);

(* When the transfer is within .1 MM of the Load Position set the indicator *)
IF ((fUAxisLoadSidePosition-0.1) <= stUAxis.NcToPlc.ActPos) AND
		(stUAxis.NcToPlc.ActPos <= (fUAxisLoadSidePosition+0.1)) THEN
	bTransferAtLoadIndicator:= TRUE;
ELSE
	bTransferAtLoadIndicator:= FALSE;
END_IF

(* When the transfer is within .1 MM of the Unload Position set the indicator *)
IF  ( (stUAxis.NcToPlc.ActPos-0.1) <= fUAxisUnloadSidePosition ) AND
	( fUAxisUnloadSidePosition <=  (stUAxis.NcToPlc.ActPos+0.1) )
THEN
	bTransferAtUnloadIndicator := TRUE;
ELSE
	bTransferAtUnloadIndicator := FALSE;
END_IF
END_PROGRAM
ACTION ChipConveyorMotorControl:
(* The Chip conveyor has a Contactor in the Power Cabinet,
	and it has a VFD on the Conveyor itself *)

(* Pull in the Chip Conveyor Contactor when the MCR is on *)

(* Chip Conveyor Contactor *)
fbChipConveyorMotorControl(
	bStart:= bMCR AND NOT( bChipConveyorMotorControlError),
	bAuxContact:= bChipConveyorMotorRunning
);

bChipConveyorOn:=fbChipConveyorMotorControl.bMSOn;
bChipConveyorMotorControlError:=fbChipConveyorMotorControl.bError;

(* VFD Output *)
(* The VFD Run command is controlled in MM_CoolantOn and MM_Coolant_Off part of Main *)
bConveyorFWDReq:=bChipConveyorMotorControl;

(* Chip Conveyor VFD Fault *)
bChipConveyorVFDFault;
END_ACTION
ACTION CycleStartControl:
fbCycleStartControl(
	bCS1:= bPB2ACycleStart OR bPB2BCycleStart,
	bCS2:= bPB3ACycleCommon OR bPB3BCycleCommon,
	bHold:= bCycleStartControlHold,
	bReset:= bCycleStartControlReset,
);

bCycleStartControlEnable:=fbCycleStartControl.bEnable;
END_ACTION
ACTION HighPressureMotorControl:
fbHighPressureMotorControl(
	bStart:=bHighPressureMotorControl ,
	bAuxContact:= bHighPressureMotorRunning
);

bHighPressureMotorOn:=fbHighPressureMotorControl.bMSOn;
bHighPressureMotorControlError:=fbHighPressureMotorControl.bError;

(* When we have a Low tank level or Overflow Switch Fault
	we shut off the High Pressure Pump imediately *)
IF bHighPressureMotorControl THEN
	IF NOT fbCoolantLevelDelayTOF.Q THEN
		bHighPressureMotorControl:=FALSE;
		nModeError:=Er_CleanTankLow;
	ELSIF NOT bCoolantTankOverflow THEN
		bHighPressureMotorControl:=FALSE;
		nModeError:=Er_CoolantOverflow;
	END_IF
END_IF
END_ACTION
ACTION HydraulicPowerUnitControl:
(* TEMPERATURE FAULT *)
IF bHydraulicTemperature OR bHydraulicPowerUnitMotorControlError THEN
	bHydraulicPowerUnitMotorControl:=FALSE;
END_IF

fbHydraulicPowerUnitMotorControl(
	bStart:=bHydraulicPowerUnitMotorControl ,
	bAuxContact:= bHydraulicPowerUnitRunning
);

bHydraulicUnitOn:=fbHydraulicPowerUnitMotorControl.bMSOn;
bHydraulicPowerUnitMotorControlError:=fbHydraulicPowerUnitMotorControl.bError;
END_ACTION
ACTION Security:
(* Set the User Level to 0 if in Auto, else to whoever has logged in *)
IF bMachineMode OR bLogoutPB THEN
	CurrentUserLevel:=0;
	sUsername:='';
	sPassword:='';
ELSIF (sUsername = sUsernameKays OR  sUsername = sUsernameKaysEngineering OR sUsername = sUsernameKaysLC) AND
		sPassword = sPasswordKays THEN
	OldUserLevel:=CurrentUserLevel;
	CurrentUserLevel:=7;
	sPassword:='';
ELSIF (sUsername = sUsernameMaint OR sUsername = sUsernameMaintLC OR
		sUsername = sUsernameMaintenance OR sUsername = sUsernameMaintenanceLC) AND
		(sPassword = sPasswordMaintenance OR sPassword = sPasswordMaint) THEN
	OldUserLevel:=CurrentUserLevel;
	CurrentUserLevel:=6;
	sPassword:='';
ELSIF (sUsername = sUsernameSuper OR sUsername = sUsernameSuperLC OR
		sUsername = sUsernameSupervisor OR sUsername = sUsernameSupervisorLC) AND
		(sPassword = sPasswordSupervisor OR sPassword = sPasswordSupervisorUC OR
		sPassword = sPasswordSuper OR sPassword = sPasswordSuperUC) THEN
	OldUserLevel:=CurrentUserLevel;
	CurrentUserLevel:=5;
	sPassword:='';
END_IF


(* Clear the User Names *)
IF (CurrentUserLevel = 5) AND
	(sUsername = sUsernameSupervisor OR sUsername = sUsernameSupervisorLC OR
	sUsername = sUsernameSuper OR sUsername = sUsernameSuperLC)
THEN
	sUsername:='';
ELSIF (CurrentUserLevel = 6) AND
	(sUsername = sUsernameMaintenance OR sUsername = sUsernameMaintenanceLC OR
	sUsername = sUsernameMaint OR sUsername = sUsernameMaintLC)
THEN
	sUsername:='';
ELSIF (CurrentUserLevel = 7) AND
	(sUsername = sUsernameKays OR sUsername = sUsernameKaysLC OR
	sUsername = sUsernameKaysEngineering)
THEN
	sUsername:='';
END_IF

(* Clear the Passwords and User Names on the screen Display boxes *)
END_ACTION
ACTION TransferPumpMotorControl:
fbTransferPumpMotorControl(
	bStart:= bTransferPumpMotorControl ,
	bAuxContact:=bTransferPumpMotorRunning
);

bTransferPumpOn:=fbTransferPumpMotorControl.bMSOn;
bTransferPumpMotorControlError:=fbTransferPumpMotorControl.bError;
END_ACTION
ACTION VFDControl:
(*The nVFDAdjustedRPM variable adjusts the entered speed command to correct for actual speed
A line like the one below should be in the Spindle Setup for the actual machine*)
(*nVFDAdjustedRPM:=LREAL_TO_UINT(nVFDControlRPM*1.0);*)

(* The Red Lion Tack's are set to 2500 for max scale *)
nRPMScaleMax:=2500;


(* Display the Tach Feedback inputs as Spindle Speeds*)
(* Side A Tacks when VFD's Enabled *)
IF bVFD_ARun THEN
	nSpindleRPM1A :=
		LREAL_TO_UDINT(nSpindleTachA1/32767.0*nRPMScaleMax);
	nSpindleRPM2A :=
		LREAL_TO_UDINT(nSpindleTachA2/32767.0*nRPMScaleMax);
	nSpindleRPM3A :=
		LREAL_TO_UDINT(nSpindleTachA3/32767.0*nRPMScaleMax);
ELSE
	nSpindleRPM1A := 0;
	nSpindleRPM2A := 0;
	nSpindleRPM3A := 0;
END_IF
(* Side B Tacks when VFD's Enabled *)
IF bVFD_BRun THEN
	nSpindleRPM1B :=
		LREAL_TO_UDINT(nSpindleTachB1/32767.0*nRPMScaleMax);
	nSpindleRPM2B :=
		LREAL_TO_UDINT(nSpindleTachB2/32767.0*nRPMScaleMax);
	nSpindleRPM3B :=
		LREAL_TO_UDINT(nSpindleTachB3/32767.0*nRPMScaleMax);
ELSE
	nSpindleRPM1B := 0;
	nSpindleRPM2B := 0;
	nSpindleRPM3B := 0;
END_IF


nVFDControlRPM:=LREAL_TO_UINT(fRPMRequest);
(* The Ratio is Motor Pulley 34 Teeth Spindle Pulley 45 teeth = 0.755556 *)
fVFDControlRatio:=(45.0/34.0);

(* 		Spindle #A1 VFD control function block *)
fbVFD_A1(
	bRun:= bVFD_ARun ,
	nRPM:= nVFDControlRPM ,
	nOverride:= 100,
	fRatio:= fVFDControlRatio ,
	bMotorDirection:= bVFDControlDirection ,
	bDataValid:= NOT(bVFD_A1DataValid),
	bReset:= bFaultResetPB OR fbCommonFautlResetTON.Q OR bAFaultResetInternal ,
	sNetId:= fbGetAMS.AxisNetId ,
	nSlaveAddr:= nVFD_A1Addr,
	bEnableDrive=> ,
	bUpToSpeed=> bVFD_A1UpToSpeed ,
	bError=> bVFD_A1Error ,
	nErrorID=> nVFD_A1ErrorID ,
	stVFDInfo=> stVFD_A1DriveInfo );

(* 		Spindle #A2 VFD control function block *)
fbVFD_A2(
	bRun:= bVFD_ARun ,
	nRPM:= nVFDControlRPM ,
	nOverride:= 100,
	fRatio:= fVFDControlRatio ,
	bMotorDirection:= bVFDControlDirection ,
	bDataValid:= NOT(bVFD_A2DataValid),
	bReset:= bFaultResetPB OR fbCommonFautlResetTON.Q OR bAFaultResetInternal ,
	sNetId:= fbGetAMS.AxisNetId ,
	nSlaveAddr:= nVFD_A2Addr,
	bEnableDrive=> ,
	bUpToSpeed=> bVFD_A2UpToSpeed ,
	bError=> bVFD_A2Error ,
	nErrorID=> nVFD_A2ErrorID ,
	stVFDInfo=> stVFD_A2DriveInfo );

(* 		Spindle #A3 VFD control function block *)
fbVFD_A3(
	bRun:= bVFD_ARun ,
	nRPM:= nVFDControlRPM ,
	nOverride:= 100,
	fRatio:= fVFDControlRatio ,
	bMotorDirection:= bVFDControlDirection ,
	bDataValid:= NOT(bVFD_A3DataValid),
	bReset:= bFaultResetPB OR fbCommonFautlResetTON.Q OR bAFaultResetInternal ,
	sNetId:= fbGetAMS.AxisNetId ,
	nSlaveAddr:= nVFD_A3Addr,
	bEnableDrive=> ,
	bUpToSpeed=> bVFD_A3UpToSpeed ,
	bError=> bVFD_A3Error ,
	nErrorID=> nVFD_A3ErrorID ,
	stVFDInfo=> stVFD_A3DriveInfo );

(* 		Spindle #B1 VFD control function block *)
fbVFD_B1(
	bRun:= bVFD_BRun ,
	nRPM:= nVFDControlRPM ,
	nOverride:= 100,
	fRatio:= fVFDControlRatio ,
	bMotorDirection:= bVFDControlDirection ,
	bDataValid:= NOT(bVFD_B1DataValid),
	bReset:= bFaultResetPB OR fbCommonFautlResetTON.Q OR bBFaultResetInternal ,
	sNetId:= fbGetAMS.AxisNetId ,
	nSlaveAddr:= nVFD_B1Addr,
	bEnableDrive=> ,
	bUpToSpeed=> bVFD_B1UpToSpeed ,
	bError=> bVFD_B1Error ,
	nErrorID=> nVFD_B1ErrorID ,
	stVFDInfo=> stVFD_B1DriveInfo );

(* 		Spindle #B2 VFD control function block *)
fbVFD_B2(
	bRun:= bVFD_BRun ,
	nRPM:= nVFDControlRPM ,
	nOverride:= 100,
	fRatio:= fVFDControlRatio ,
	bMotorDirection:= bVFDControlDirection ,
	bDataValid:= NOT(bVFD_B2DataValid),
	bReset:= bFaultResetPB OR fbCommonFautlResetTON.Q OR bBFaultResetInternal ,
	sNetId:= fbGetAMS.AxisNetId ,
	nSlaveAddr:= nVFD_B2Addr,
	bEnableDrive=> ,
	bUpToSpeed=> bVFD_B2UpToSpeed ,
	bError=> bVFD_B2Error ,
	nErrorID=> nVFD_B2ErrorID ,
	stVFDInfo=> stVFD_B2DriveInfo );

(* 		Spindle #B3 VFD control function block *)
fbVFD_B3(
	bRun:= bVFD_BRun ,
	nRPM:= nVFDControlRPM ,
	nOverride:= 100,
	fRatio:= fVFDControlRatio ,
	bMotorDirection:= bVFDControlDirection ,
	bDataValid:= NOT(bVFD_B3DataValid),
	bReset:= bFaultResetPB OR fbCommonFautlResetTON.Q OR bBFaultResetInternal ,
	sNetId:= fbGetAMS.AxisNetId ,
	nSlaveAddr:= nVFD_B3Addr,
	bEnableDrive=> ,
	bUpToSpeed=> bVFD_B3UpToSpeed ,
	bError=> bVFD_B3Error ,
	nErrorID=> nVFD_B3ErrorID ,
	stVFDInfo=> stVFD_B3DriveInfo );

(* Get the AMS Net ID of the CX TwinCAT when the MCC_V Contactor Pulled In *)
fbGetAMS(
	sNetId:='' ,
	iAxisId:=1 ,
	bExecute:=bMCC_V );
END_ACTION
ACTION Z_AxisControl:
(* Turn on MC_Power when Hard Enable is ON *)
bZAAxisPower := bAServoEnable;

fbZAAxisPower(
	Enable:=bZAAxisPower ,
	Enable_Positive:=bZAAxisPower ,
	Enable_Negative:=bZAAxisPower ,
	Override:=100 ,
	BufferMode:=MC_Aborting ,
	Axis:=stZAAxis );

fbZAAxisSetZero(
	Execute:=bZAAxisSetZero,
	Position:=0.0,
	HomingMode:=MC_Direct,
	Axis:=stZAAxis );

fbZAAxisMove(
	Execute:= bZAAxisMove ,
	Position:= fZAMovePosition ,
	Velocity:= fZAMoveVelocity ,
	Acceleration:= 0 ,
	Deceleration:= 0,
	Jerk := 0,
	BufferMode:=MC_Aborting ,
	Axis := stZAAxis );

(* When the Axis Stop is done, then turn off the enable
	Must be above the Command so the done bit will be true for a scan *)
IF bZAStop AND fbZAAxisStop.Done THEN
	bZAStop:=FALSE;
END_IF
fbZAAxisStop(
	Execute := bZAStop,
	Deceleration := 0,
	Jerk := 0,
	Axis := stZAAxis );

fbZAAxisMCReset(
	Execute:=bZAMCResetRequest ,
	Axis:=stZAAxis );

fbZAAxisDriveReset(
	NetId:='' ,
	Execute:=bZWADriveResetRequest ,
	Timeout:=t#10s ,
	Axis:= stZAAxis, );

stZAAxis.ReadStatus();

(* If one of the ZA Axis overtravel limit switches is made, then turn on the bit that allows
Movement off of the limit switchs *)
IF NOT(DriveZAWAdinputs.0) OR NOT(DriveZAWAdinputs.1) THEN
	bZADeCtrlEnable:=TRUE;
ELSE
	bZADeCtrlEnable:=FALSE;
END_IF
stZAAxis.PlcToNc.ControlDWord :=
AxisSetAcceptBlockedDriveSignal(stZAAxis.PlcToNc.ControlDWord,
	bEnable:= bZADeCtrlEnable );

(* If a Drive reset was requested then when the Drive Reset is done we want to do a MC Reset of the NC Axis *)
IF bZWADriveResetRequest AND (NOT (fbZAAxisDriveReset.Busy) OR  fbZAAxisDriveReset.Error) THEN
	bZAMCResetRequest:=TRUE;
(* Else if the MC Reset is on when when the Drive Reset it busy it must have stuck on so we want to turn it off *)
ELSIF bZWADriveResetRequest AND fbZAAxisDriveReset.Busy AND bZAMCResetRequest THEN
	bZAMCResetRequest:=FALSE;
END_IF
IF fbZAAxisMCReset.Done THEN
	bZAMCResetRequest:=FALSE;
	bZWADriveResetRequest:=FALSE;
END_IF

(* 			Z Axis Side B 			*)

(* Turn on MC_Power when Hard Enable is ON *)
bZBAxisPower := bBServoEnable;

fbZBAxisPower(
	Enable:=bZBAxisPower ,
	Enable_Positive:=bZBAxisPower ,
	Enable_Negative:=bZBAxisPower ,
	Override:=100 ,
	BufferMode:=MC_Aborting ,
	Axis:=stZBAxis );

fbZBAxisSetZero(
	Execute:=bZBAxisSetZero,
	Position:=0.0,
	HomingMode:=MC_Direct,
	Axis:=stZBAxis );

fbZBAxisMove(
	Execute:= bZBAxisMove ,
	Position:= fZBMovePosition ,
	Velocity:= fZBMoveVelocity ,
	Acceleration:= 0 ,
	Deceleration:= 0,
	Jerk := 0,
	BufferMode:=MC_Aborting ,
	Axis := stZBAxis );

(* When the Axis Stop is done, then turn off the enable
	Must be above the Command so the done bit will be true for a scan *)
IF bZBStop AND fbZBAxisStop.Done THEN
	bZBStop:=FALSE;
END_IF
fbZBAxisStop(
	Execute := bZBStop,
	Deceleration := 0,
	Jerk := 0,
	Axis := stZBAxis );

fbZBAxisMCReset(
	Execute:=bZBMCResetRequest ,
	Axis:=stZBAxis );

fbZBAxisDriveReset(
	NetId:='' ,
	Execute:=bZWBDriveResetRequest ,
	Timeout:=t#10s ,
	Axis:= stZBAxis, );

stZBAxis.ReadStatus();

(* If one of the ZB Axis overtravel limit switches is made, then turn on the bit that allows
Movement off of the limit switchs *)
IF NOT(DriveZBWBdinputs.0) OR NOT(DriveZBWBdinputs.1) THEN
	bZBDeCtrlEnable:=TRUE;
ELSE
	bZBDeCtrlEnable:=FALSE;
END_IF
stZBAxis.PlcToNc.ControlDWord :=
AxisSetAcceptBlockedDriveSignal(stZBAxis.PlcToNc.ControlDWord,
	bEnable:= bZBDeCtrlEnable );

(* If a Drive reset was requested then when the Drive Reset is done we want to do a MC Reset of the NC Axis *)
IF bZWBDriveResetRequest AND (NOT (fbZBAxisDriveReset.Busy) OR  fbZBAxisDriveReset.Error) THEN
	bZBMCResetRequest:=TRUE;
(* Else if the MC Reset is on when when the Drive Reset it busy it must have stuck on so we want to turn it off *)
ELSIF bZWBDriveResetRequest AND fbZBAxisDriveReset.Busy AND bZBMCResetRequest THEN
	bZBMCResetRequest:=FALSE;
END_IF
IF fbZBAxisMCReset.Done THEN
	bZBMCResetRequest:=FALSE;
	bZWBDriveResetRequest:=FALSE;
END_IF
END_ACTION

(* POU Function Blocks/FB_MotorStarter, ST *)
FUNCTION_BLOCK FB_MotorStarter
(*
	Author:		Brandon Snell 	Date:		01.23.2008
	Modified:		Ron Poehlmann	10-23-2014  Removed Error ID
*)
VAR_INPUT
	bStart: BOOL := FALSE;						(* 	Level Trigger to Turn On Motor Starter, Edge Triggers Timer *)
	bAuxContact: BOOL :=TRUE;					(* 	Check To Ensure Motor Starter Is On, If No Auxilary Contact
														Present This Shall Remain TRUE *)
END_VAR
VAR_OUTPUT
	bMSOn: BOOL :=FALSE;						(* 	Simply Turns On When bStart is Level HIGH, Errors Will Turn Output Off,
														bStart must be cycled because positive edge bStart Resets bError *)
	bError: BOOL :=FALSE;						(* 	Bit telling on the motor starter failure *)
END_VAR
VAR
	fbStartRTrig: R_TRIG;
	bStartTime: BOOL := FALSE;
	fbDelayTimer: TON;
	fbStartFTrig: F_TRIG;
END_VAR
(*
	fbStartRTrig finds the rising edge of bStart in order
	to initialize the delay timer 
*)
fbStartRTrig(CLK:=bStart , Q=> );

(*
	fbStartFTrig finds the falling edge of bStart used to
	reset the current error state of the function block 
*)
fbStartFTrig(CLK:=bStart , Q=> );

(*
	fbDelayTimer is used to allow for possible bounce
	in auxilary contact closure
*)
fbDelayTimer(IN:=bStartTime , PT:=t#1s500ms , Q=> , ET=> );

(*
	Reset Error State Returning To Initial State
*)
IF fbStartFTrig.Q THEN
	bError:=FALSE;
END_IF

(*
	Initialize Delay Timer Jumping To Run State #1
*)
IF fbStartRTrig.Q THEN
	bStartTime:=TRUE;
END_IF

(*
	Set Error For Motor Starter Jumping to Error State
	If bAuxContact does not fail to close then Jumping to Run State #2
*)
IF bStart AND NOT(bAuxContact) AND fbDelayTimer.Q THEN
	bError:=TRUE;
END_IF



(*
	Turn On Motor Starter Level HIGH bStart
*)
IF bStart AND NOT(bError) THEN
	bMSOn:=TRUE;
ELSE
	bMSOn:=FALSE;
END_IF

(*
	Prepare Timer For Edge Triggered Start
*)
IF NOT(bStart) THEN
	bStartTime:=FALSE;
END_IF
END_FUNCTION_BLOCK

(* POU Function Blocks/FB_CycleStart, ST *)
FUNCTION_BLOCK FB_CycleStart
VAR
	fbTimerOne: TON; 			(* 	The timer will only expire if one or the other is pressed by itself *)
	bContinue: BOOL := FALSE; 	(* 	This will be set to TRUE at the event that cycle start has been cleared to
										continue without CS1 AND CS2 TRUE *)
END_VAR
VAR_INPUT
	bCS1: BOOL := FALSE; 		(* 	Cycle Start #1 *)
	bCS2: BOOL := FALSE; 		(* 	Cycle Start #2 *)
	bHold: BOOL := FALSE; 		(* 	This should go TRUE at the point that it has been deemed safe to continue operation *)
	bReset: BOOL := FALSE; 		(* 	Reset all variables to FALSE *)
END_VAR
VAR_OUTPUT
	bEnable: BOOL := FALSE; 	(* 	If conditions are met this will be TRUE upon release of both cycle starts *)
END_VAR
(* Internally reset this function back to the initial state *)
	IF bReset THEN
		bEnable:=FALSE;
		bContinue:=FALSE;
	END_IF;

(* Set fbTimerOne if and only if either CS1 is true OR CS2 is true but not both *)
	fbTimerOne(IN:= bCS1 XOR bCS2 , PT:= T#500ms , Q=> , ET=> );

(* Ensure Anti-Tie Down and safety is ensured *)
	IF bCS1 AND bCS2 AND NOT fbTimerOne.Q THEN
		bEnable:=TRUE;
	ELSIF bContinue THEN
		bEnable:=TRUE;
	ELSE
		bEnable:=FALSE;
	END_IF;

(* Once the block has been issued hold then CS1 AND CS2 can be released *)
	IF bCS1 AND bCS2 AND NOT fbTimerOne.Q AND bHold THEN
		bContinue:=TRUE;
	END_IF;
END_FUNCTION_BLOCK

(* POU Programs/DEMO, LD *)
PROGRAM DEMO
VAR
	ComOnTON: TON;
	ComOffTON: TON;
END_VAR
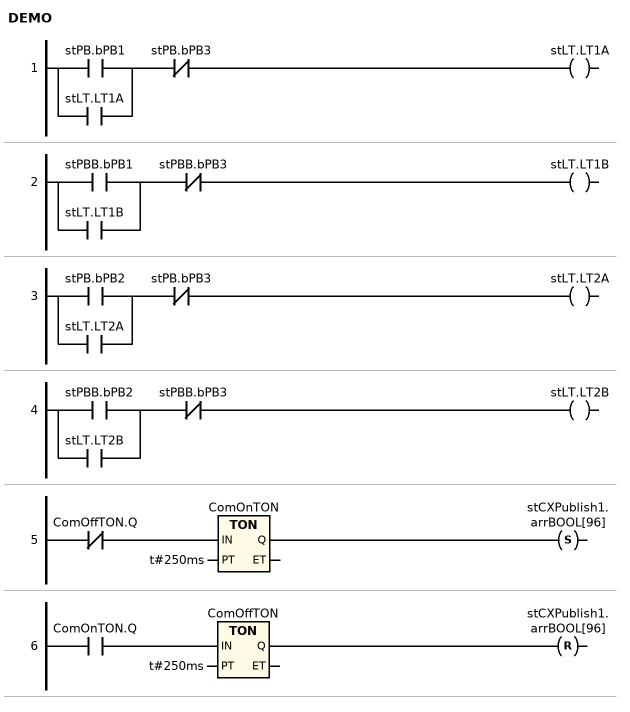
_LD_ (* Ladder Diagram *)
NETWORK 1
	{ [stPB.bPB1] | [stLT.LT1A] } - [/stPB.bPB3] --- (stLT.LT1A)
NETWORK 2
	{ [stPBB.bPB1] | [stLT.LT1B] } - [/stPBB.bPB3] --- (stLT.LT1B)
NETWORK 3
	{ [stPB.bPB2] | [stLT.LT2A] } - [/stPB.bPB3] --- (stLT.LT2A)
NETWORK 4
	{ [stPBB.bPB2] | [stLT.LT2B] } - [/stPBB.bPB3] --- (stLT.LT2B)
NETWORK 5
	[/ComOffTON.Q] - ComOnTON:TON(IN: *, PT: t#250ms) --- (S stCXPublish1.arrBOOL[96])
NETWORK 6
	[ComOnTON.Q] - ComOffTON:TON(IN: *, PT: t#250ms) --- (R stCXPublish1.arrBOOL[96])
_END_LD_
(* the same logic as Structured Text *)
(* Network 1 *)
stLT.LT1A := (stPB.bPB1 OR stLT.LT1A) AND NOT stPB.bPB3;
(* Network 2 *)
stLT.LT1B := (stPBB.bPB1 OR stLT.LT1B) AND NOT stPBB.bPB3;
(* Network 3 *)
stLT.LT2A := (stPB.bPB2 OR stLT.LT2A) AND NOT stPB.bPB3;
(* Network 4 *)
stLT.LT2B := (stPBB.bPB2 OR stLT.LT2B) AND NOT stPBB.bPB3;
(* Network 5 *)
ComOnTON(IN := NOT ComOffTON.Q, PT := t#250ms);
IF ComOnTON.Q THEN stCXPublish1.arrBOOL[96] := TRUE; END_IF;
(* Network 6 *)
ComOffTON(IN := ComOnTON.Q, PT := t#250ms);
IF ComOffTON.Q THEN stCXPublish1.arrBOOL[96] := FALSE; END_IF;
END_PROGRAM

(* POU Programs/P_FaultChecking, ST *)
PROGRAM P_FaultChecking
VAR
	nSpindleSpeedVariationMax: UDINT := 0;
	nSpindleSpeedVariationMin: UDINT := 0;
	bFaultResetRequested: BOOL := FALSE;

	(* Flow Monitors *)
	bHighFlow1A: BOOL := FALSE;
	bLowFlow1A: BOOL := FALSE;
	bHighFlow2A: BOOL := FALSE;
	bLowFlow2A: BOOL := FALSE;
	bHighFlow3A: BOOL := FALSE;
	bLowFlow3A: BOOL := FALSE;
	bHighFlow1B: BOOL := FALSE;
	bLowFlow1B: BOOL := FALSE;
	bHighFlow2B: BOOL := FALSE;
	bLowFlow2B: BOOL := FALSE;
	bHighFlow3B: BOOL := FALSE;
	bLowFlow3B: BOOL := FALSE;
	fbFlowAverageTimer1AHIGH: TON;
	fbFlowAverageTimer1ALOW: TON;
	fbFlowAverageTimer2AHIGH: TON;
	fbFlowAverageTimer2ALOW: TON;
	fbFlowAverageTimer3AHIGH: TON;
	fbFlowAverageTimer3ALOW: TON;
	fbFlowAverageTimer1BHIGH: TON;
	fbFlowAverageTimer1BLOW: TON;
	fbFlowAverageTimer2BHIGH: TON;
	fbFlowAverageTimer2BLOW: TON;
	fbFlowAverageTimer3BHIGH: TON;
	fbFlowAverageTimer3BLOW: TON;
	fbCoolantOnDelayTON: TON;

	(* Filter Fault Variables *)
	nDirtyCount1: UDINT := 0;
	nDirtyCount2: UDINT := 0;
	nDirtyCount3: UDINT := 0;
	nDirtyCount4: UDINT := 0;
	bFilter1Timer: BOOL := FALSE;
	bFilter2Timer: BOOL := FALSE;
	bFilter3Timer: BOOL := FALSE;
	bFilter4Timer: BOOL := FALSE;

(*Timers and Triggers *)
	fbCycleCommonTimeout: TON;
	fbFilter1Timer: TON;
	fbFilter2Timer: TON;
	fbFilter3Timer: TON;
	fbFilter4Timer: TON;

	fbLowPressureFaultADelay: TON;
	fbLowPressureFaultBDelay: TON;
	fbCoolantStartTimer: TON;
	fbCoolantTempFaultTON: TON;
	fbCoolantTempWarningTON: TON;
	fbHydraulicSystemOnTON: TON;
	fbHydraulicFluidLowTON: TON;
	fbLubePressureTON: TON;				(* Timer to fault with low lube pressure *)
	fbLubeLevelCheckRTrig: R_TRIG;		(* Check for Low Lube Level at end of Cycle *)
	nLubeLevelLowCount: INT :=0;			(* Count the number of cycles with Low Lube for Fault *)

	fbServoAThrustMaxDelayTON: TON;
	fbServoBThrustMaxDelayTON: TON;
	fbALoadFaultDelay: TON;				(* Side A Spindle Load Fault Delay Timer *)
	fbBLoadFaultDelay: TON;				(* Side B Spindle Load Fault Delay Timer *)
	(* Spindle Speed Timers *)
	fbASpeedDelayTimer: TON;
	fbSpeedVariationTimer1ALOW: TON;
	fbSpeedVariationTimer1AHIGH: TON;
	fbSpeedVariationTimer2ALOW: TON;
	fbSpeedVariationTimer2AHIGH: TON;
	fbSpeedVariationTimer3ALOW: TON;
	fbSpeedVariationTimer3AHIGH: TON;
	fbBSpeedDelayTimer: TON;
	fbSpeedVariationTimer1BLOW: TON;
	fbSpeedVariationTimer1BHIGH: TON;
	fbSpeedVariationTimer2BLOW: TON;
	fbSpeedVariationTimer2BHIGH: TON;
	fbSpeedVariationTimer3BLOW: TON;
	fbSpeedVariationTimer3BHIGH: TON;
(* Fault Program Variables *)
	nFaultState: UDINT := 0;
	nHistoryStep : USINT := 1;
	arrFaultHistoryTemp: ARRAY[1..80] OF STRING (52) := 80('');
	arrFaultWarningCurrent : ARRAY[0..9] OF STRING (52) := 10('');
	fbFaultResetWatchdog: TON;	(* Make sure we do not get stuck in the Fault Reset step *)
	nCurrent : USINT := 0;
	nUnStored : USINT := 0;

	fbInternalResetTON: TON;				(* A time delay to trigger turning off the Internal Reset *)
	fbMCRJustOnTON: TON;				(* A time delay of the MCR just turned on *)
END_VAR
fbCycleCommonTimeout(IN:= bPB2ACycleStart OR bPB3ACycleCommon OR bPB2BCycleStart OR bPB3BCycleCommon , PT:=t#10s);
(* When the Common PB is made for 1/2 second without the Cycle Start PB then Trigger a Fault Reset *)
fbCommonFautlResetTON(IN:= (bPB3ACycleCommon AND NOT(bPB2ACycleStart)) OR
	(bPB3BCycleCommon AND NOT(bPB2BCycleStart)) , PT:=t#500ms );
fbFilter1Timer(IN:= bFilter1Timer , PT:=t#40s);
fbFilter2Timer(IN:= bFilter2Timer , PT:=t#40s);
fbFilter3Timer(IN:= bFilter3Timer , PT:=t#40s);
fbFilter4Timer(IN:= bFilter4Timer , PT:=t#40s);
fbCoolantStartTimer(IN:= MAIN.bTransferPumpMotorControl,	PT:=t#15s);
fbCoolantTempFaultTON(IN:=bCoolantTempFault, PT:=t#100ms);
fbCoolantTempWarningTON(IN:=bCoolantTempWarning, PT:=t#100ms);
fbCoolantOnDelayTON(IN:=bACoolantSolenoid  OR bBCoolantSolenoid,PT:=t#1500ms);
(* Flow Monitor Timers *)
fbFlowAverageTimer1ALOW(IN:=bLowFlow1A AND bACoolantSolenoid , PT:=t#1000ms);
fbFlowAverageTimer1AHIGH(IN:=bHighFlow1A AND bACoolantSolenoid , PT:=t#1000ms);
fbFlowAverageTimer2ALOW(IN:=bLowFlow2A AND bACoolantSolenoid , PT:=t#1000ms);
fbFlowAverageTimer2AHIGH(IN:=bHighFlow2A AND bACoolantSolenoid , PT:=t#1000ms);
fbFlowAverageTimer3ALOW(IN:=bLowFlow3A AND bACoolantSolenoid , PT:=t#1000ms);
fbFlowAverageTimer3AHIGH(IN:=bHighFlow3A AND bACoolantSolenoid , PT:=t#1000ms);

fbFlowAverageTimer1BLOW(IN:=bLowFlow1B AND bBCoolantSolenoid , PT:=t#1000ms);
fbFlowAverageTimer1BHIGH(IN:=bHighFlow1B AND bBCoolantSolenoid , PT:=t#1000ms);
fbFlowAverageTimer2BLOW(IN:=bLowFlow2B AND bBCoolantSolenoid , PT:=t#1000ms);
fbFlowAverageTimer2BHIGH(IN:=bHighFlow2B AND bBCoolantSolenoid , PT:=t#1000ms);
fbFlowAverageTimer3BLOW(IN:=bLowFlow3B AND bBCoolantSolenoid , PT:=t#1000ms);
fbFlowAverageTimer3BHIGH(IN:=bHighFlow3B AND bBCoolantSolenoid , PT:=t#1000ms);

fbServoAThrustMaxDelayTON(IN:=nServoAThrustDisplay>nServoThrustMax, PT:=t#200ms);
fbServoBThrustMaxDelayTON(IN:=nServoBThrustDisplay>nServoThrustMax, PT:=t#200ms);

(* Side A Spindle Speed Delay *)
(*	Calculate Comparison Variables *)
nSpindleSpeedVariationMax:=(MAIN.nVFDControlRPM+199);
nSpindleSpeedVariationMin:=(MAIN.nVFDControlRPM-199);
fbASpeedDelayTimer(IN:=bVFD_A1UpToSpeed AND bVFD_A2UpToSpeed AND bVFD_A3UpToSpeed,
	PT:=LREAL_TO_TIME(5+stVFD_A1DriveInfo.fAccelerationTime*1000));
fbSpeedVariationTimer1ALOW(IN:=nSpindleRPM1A<nSpindleSpeedVariationMin ,PT:=t#250ms);
fbSpeedVariationTimer1AHIGH(IN:=nSpindleRPM1A>nSpindleSpeedVariationMax ,PT:=t#250ms);
fbSpeedVariationTimer2ALOW(IN:=nSpindleRPM2A<nSpindleSpeedVariationMin ,PT:=t#250ms);
fbSpeedVariationTimer2AHIGH(IN:=nSpindleRPM2A>nSpindleSpeedVariationMax ,PT:=t#250ms);
fbSpeedVariationTimer3ALOW(IN:=nSpindleRPM3A<nSpindleSpeedVariationMin ,PT:=t#250ms);
fbSpeedVariationTimer3AHIGH(IN:=nSpindleRPM3A>nSpindleSpeedVariationMax ,PT:=t#250ms);
(* Side A Spindle Speed Delay *)
fbBSpeedDelayTimer(IN:=bVFD_B1UpToSpeed AND bVFD_B2UpToSpeed AND bVFD_B3UpToSpeed,
	PT:=LREAL_TO_TIME(5+stVFD_B1DriveInfo.fAccelerationTime*1000));
fbSpeedVariationTimer1BLOW(IN:=nSpindleRPM1B<nSpindleSpeedVariationMin ,PT:=t#250ms);
fbSpeedVariationTimer1BHIGH(IN:=nSpindleRPM1B>nSpindleSpeedVariationMax ,PT:=t#250ms);
fbSpeedVariationTimer2BLOW(IN:=nSpindleRPM2B<nSpindleSpeedVariationMin ,PT:=t#250ms);
fbSpeedVariationTimer2BHIGH(IN:=nSpindleRPM2B>nSpindleSpeedVariationMax ,PT:=t#250ms);
fbSpeedVariationTimer3BLOW(IN:=nSpindleRPM3B<nSpindleSpeedVariationMin ,PT:=t#250ms);
fbSpeedVariationTimer3BHIGH(IN:=nSpindleRPM3B>nSpindleSpeedVariationMax ,PT:=t#250ms);
(*	Spindle Load Delay *)
fbALoadFaultDelay(
	IN:= bVFD_A1UpToSpeed AND bVFD_A2UpToSpeed AND bVFD_A3UpToSpeed ,
	PT:=t#1500ms);
fbBLoadFaultDelay(
	IN:= bVFD_B1UpToSpeed AND bVFD_B2UpToSpeed AND bVFD_B3UpToSpeed ,
	PT:=t#1500ms);

(*	Flow Fault Helper *)
(* SIDE A *)
IF ( fCoolantFlow1ADisplay<fCoolantFlowMin ) AND bACoolantSolenoid THEN
	bLowFlow1A:=TRUE;
ELSE
	bLowFlow1A:=FALSE;
END_IF
IF ( fCoolantFlow1ADisplay>fCoolantFlowMax ) AND bACoolantSolenoid THEN
	bHighFlow1A:=TRUE;
ELSE
	bHighFlow1A:=FALSE;
END_IF
IF ( fCoolantFlow2ADisplay<fCoolantFlowMin ) AND bACoolantSolenoid THEN
	bLowFlow2A:=TRUE;
ELSE
	bLowFlow2A:=FALSE;
END_IF
IF ( fCoolantFlow2ADisplay>fCoolantFlowMax ) AND bACoolantSolenoid THEN
	bHighFlow2A:=TRUE;
ELSE
	bHighFlow2A:=FALSE;
END_IF
IF ( fCoolantFlow3ADisplay<fCoolantFlowMin ) AND bACoolantSolenoid THEN
	bLowFlow3A:=TRUE;
ELSE
	bLowFlow3A:=FALSE;
END_IF
IF ( fCoolantFlow3ADisplay>fCoolantFlowMax ) AND bACoolantSolenoid THEN
	bHighFlow3A:=TRUE;
ELSE
	bHighFlow3A:=FALSE;
END_IF

(* SIDE B *)
IF ( fCoolantFlow1BDisplay<fCoolantFlowMin ) AND bBCoolantSolenoid THEN
	bLowFlow1B:=TRUE;
ELSE
	bLowFlow1B:=FALSE;
END_IF
IF ( fCoolantFlow1BDisplay>fCoolantFlowMax ) AND bBCoolantSolenoid THEN
	bHighFlow1B:=TRUE;
ELSE
	bHighFlow1B:=FALSE;
END_IF
IF ( fCoolantFlow2BDisplay<fCoolantFlowMin ) AND bBCoolantSolenoid THEN
	bLowFlow2B:=TRUE;
ELSE
	bLowFlow2B:=FALSE;
END_IF
IF ( fCoolantFlow2BDisplay>fCoolantFlowMax ) AND bBCoolantSolenoid THEN
	bHighFlow2B:=TRUE;
ELSE
	bHighFlow2B:=FALSE;
END_IF
IF ( fCoolantFlow3BDisplay<fCoolantFlowMin ) AND bBCoolantSolenoid THEN
	bLowFlow3B:=TRUE;
ELSE
	bLowFlow3B:=FALSE;
END_IF
IF ( fCoolantFlow3BDisplay>fCoolantFlowMax ) AND bBCoolantSolenoid THEN
	bHighFlow3B:=TRUE;
ELSE
	bHighFlow3B:=FALSE;
END_IF


(*	Filter Fault Helper *)
IF NOT(bFilter1Dirty) THEN
	nDirtyCount1:=0;
ELSIF bFilter1Dirty AND NOT(bFilter1Timer) THEN
	bFilter1Timer:=TRUE;
END_IF
IF NOT(bFilter2Dirty) THEN
	nDirtyCount2:=0;
ELSIF bFilter2Dirty AND NOT(bFilter2Timer) THEN
	bFilter2Timer:=TRUE;
END_IF
IF NOT(bFilter3Dirty) THEN
	nDirtyCount3:=0;
ELSIF bFilter3Dirty AND NOT(bFilter3Timer) THEN
	bFilter3Timer:=TRUE;
END_IF
IF NOT(bFilter4Dirty) THEN
	nDirtyCount4:=0;
ELSIF bFilter4Dirty AND NOT(bFilter4Timer) THEN
	bFilter4Timer:=TRUE;
END_IF

fbCoolantLevelDelayTOF(IN:=bCleanTankLevel, PT:=t#2s);
(*	Hydraulic Unit On *)
fbHydraulicSystemOnTON(IN:=bHydraulicPowerUnitRunning , PT:=t#1s);
(*	Hydraulic Unit Fluid Level Low Delay *)
fbHydraulicFluidLowTON(IN:=NOT(bHydraulicSystemLevel)
	AND bHydraulicPowerUnitRunning, PT:=t#5s);
(*	Lube Pressure Delayed *)
fbLubePressureTON(IN:= bWayLubePump AND NOT(bLubePressure),
	PT:=t#30m);
(*	Check for Low Lube when at end of cycle *)
fbLubeLevelCheckRTrig(CLK:=(nAutoCycleStep=AC_Unclamp) AND (NOT bLubeLevel));
(* 	Count up when Lube Level is low at the end of a cycle *)
IF fbLubeLevelCheckRTrig.Q THEN
	nLubeLevelLowCount:= nLubeLevelLowCount+1;
(* Reset Count if Lube Level Restored *)
ELSIF bLubeLevel THEN
	nLubeLevelLowCount:=0;
END_IF
(*	Coolant Pressure Low - Side A*)
fbLowPressureFaultADelay(IN:=bACoolantSolenoid AND NOT bACoolantPressure, PT:=t#2000ms);
(*	Coolant Pressure Low - Side B*)
fbLowPressureFaultBDelay(IN:=bBCoolantSolenoid AND NOT bBCoolantPressure, PT:=t#2000ms);

(* Array Assignments:
	nActiveFaults[1] => standard machine faults
	nActiveFaults[2] => Side A Faults
	nActiveFaults[3] => Side B Faults
	nActiveFaults[4] => Specific Faults Like Filter that Do not shut off the machines	*)

CASE nFaultState OF
	0:	(* Check for any faults *)

		IF nActiveFaults[1].0=0 AND NOT( bMCR) THEN
			nActiveFaults[1].0:=1;
			IF (nFaultArrayIndex<=5) THEN
				arrFaultMessage[nFaultArrayIndex]:='F001 - Machine has been in the ESTOP state';
				arrFaultWarningCurrent[nCurrent]:='F001 - Machine has been in the ESTOP state';
				nFaultArrayIndex:=nFaultArrayIndex+1;
				nCurrent:=nCurrent+1;
			END_IF
		END_IF

		IF nActiveFaults[1].1=0 AND bInCycle
				AND (NOT(bPB4ADrillReturn) OR NOT(bPB4BDrillReturn))
		THEN
			nActiveFaults[1].1:=1;
			IF (nFaultArrayIndex<=5) THEN
				arrFaultMessage[nFaultArrayIndex]:='F002 - Drill Return Activated';
				arrFaultWarningCurrent[nCurrent]:='F002 - Drill Return Activated';
				nFaultArrayIndex:=nFaultArrayIndex+1;
				nCurrent:=nCurrent+1;
			END_IF
		END_IF

		IF nActiveFaults[1].2=0 AND MAIN.bHighPressureMotorControlError AND MAIN.bHighPressureMotorControl THEN
			nActiveFaults[1].2:=1;
			IF (nFaultArrayIndex<=5) THEN
				arrFaultMessage[nFaultArrayIndex]:='F003 - High Pressure Motor Starter Failed';
				arrFaultWarningCurrent[nCurrent]:='F003 - High Pressure Motor Starter Failed';
				nFaultArrayIndex:=nFaultArrayIndex+1;
				nCurrent:=nCurrent+1;
			END_IF
		END_IF

		IF nActiveFaults[1].3=0 AND MAIN.bTransferPumpMotorControlError AND MAIN.bTransferPumpMotorControl THEN
			nActiveFaults[1].3:=1;
			IF (nFaultArrayIndex<=5) THEN
				arrFaultMessage[nFaultArrayIndex]:='F004 - Transfer Pump Motor Starter Failed';
				arrFaultWarningCurrent[nCurrent]:='F004 - Transfer Pump Motor Starter Failed';
				nFaultArrayIndex:=nFaultArrayIndex+1;
				nCurrent:=nCurrent+1;
			END_IF
		END_IF

		IF nActiveFaults[1].4=0 AND (bInCycle OR bSetup) AND NOT(bProx313) THEN
			nActiveFaults[1].4:=1;
			IF (nFaultArrayIndex<=5) THEN
				arrFaultMessage[nFaultArrayIndex]:='F005 - Fixture Door Open Side B';
				arrFaultWarningCurrent[nCurrent]:='F005 - Fixture Door Open Side B';
				nFaultArrayIndex:=nFaultArrayIndex+1;
				nCurrent:=nCurrent+1;
			END_IF
		END_IF

		IF nActiveFaults[1].5=0 AND ( (NOT(fbCoolantLevelDelayTOF.Q)
			AND fbCoolantStartTimer.Q) OR
			nModeError=Er_CleanTankLow )
		 THEN
			nActiveFaults[1].5:=1;
			IF nModeError=Er_CleanTankLow THEN
				nModeError:=Er_NoModeError;
			END_IF
			IF (nFaultArrayIndex<=5) THEN
				arrFaultMessage[nFaultArrayIndex]:='F006 - Coolant Tank Level Low';
				arrFaultWarningCurrent[nCurrent]:='F006 - Coolant Tank Level Low';
				nFaultArrayIndex:=nFaultArrayIndex+1;
				nCurrent:=nCurrent+1;
			END_IF
		END_IF

		IF nActiveFaults[1].6=0 AND fbCoolantTempFaultTON.Q THEN
			nActiveFaults[1].6:=1;
			IF (nFaultArrayIndex<=5) THEN
				arrFaultMessage[nFaultArrayIndex]:='F007 - Coolant Temperature Fault';
				arrFaultWarningCurrent[nCurrent]:='F007 - Coolant Temperature Fault';
				nFaultArrayIndex:=nFaultArrayIndex+1;
				nCurrent:=nCurrent+1;
			END_IF
		END_IF

		IF nActiveFaults[1].7=0 AND nModeError=Er_CoolantOverflow THEN
			nActiveFaults[1].7:=1;
			nModeError:=Er_NoModeError;
			IF (nFaultArrayIndex<=5) THEN
				arrFaultMessage[nFaultArrayIndex]:='F008 - Coolant Tank Overflow';
				arrFaultWarningCurrent[nCurrent]:='F008 - Coolant Tank Overflow';
				nFaultArrayIndex:=nFaultArrayIndex+1;
				nCurrent:=nCurrent+1;
			END_IF
		END_IF

		IF nActiveFaults[1].8=0 AND MAIN.bHydraulicPowerUnitMotorControlError
			AND MAIN.bHydraulicPowerUnitMotorControl
		THEN
			nActiveFaults[1].8:=1;
			IF (nFaultArrayIndex<=5) THEN
				arrFaultMessage[nFaultArrayIndex]:='F009 - Hydraulic Power Unit Motor Starter Failed';
				arrFaultWarningCurrent[nCurrent]:='F009 - Hydraulic Power Unit Motor Starter Failed';
				nFaultArrayIndex:=nFaultArrayIndex+1;
				nCurrent:=nCurrent+1;
			END_IF
		END_IF

		IF nActiveFaults[1].9=0 AND nModeError=Er_AMUnclampTimeout THEN
			nActiveFaults[1].9:=1;
			nModeError:=Er_NoModeError;
			IF (nFaultArrayIndex<=5) THEN
				arrFaultMessage[nFaultArrayIndex]:='F010 - Part Unclamp Timeout';
				arrFaultWarningCurrent[nCurrent]:='F010 - Part Unclamped Timeout';
				nFaultArrayIndex:=nFaultArrayIndex+1;
				nCurrent:=nCurrent+1;
			END_IF
		END_IF

		(* During SETUP Mode an Error occurred with the Clamping *)
		IF nActiveFaults[1].10=0 AND nModeError=Er_SetupError THEN
			nActiveFaults[1].10:=1;
			IF (nFaultArrayIndex<=5) THEN
				CASE nSetupErrorID OF
				1:
					arrFaultMessage[nFaultArrayIndex]:='F011a - Parts Missing';
					arrFaultWarningCurrent[nCurrent]:='F011a - Parts Missing';
				2:
					arrFaultMessage[nFaultArrayIndex]:='F011b - Clamp PS OFF';
					arrFaultWarningCurrent[nCurrent]:='F011b - Clamp PS OFF';
				3:
					arrFaultMessage[nFaultArrayIndex]:='F011c - Unclamp PS ON';
					arrFaultWarningCurrent[nCurrent]:='F011c - Unclamp PS ON';
				END_CASE
				nFaultArrayIndex:=nFaultArrayIndex+1;
				nCurrent:=nCurrent+1;
			END_IF
			nModeError:=Er_NoModeError;
			nSetupErrorID:=0;
		END_IF

		IF nActiveFaults[1].11=0 AND (bInCycle OR bSetup) AND NOT(bProx310) THEN
			nActiveFaults[1].11:=1;
			IF (nFaultArrayIndex<=5) THEN
				arrFaultMessage[nFaultArrayIndex]:='F012 - Tool Change Door Open Side A';
				arrFaultWarningCurrent[nCurrent]:='F012 - Tool Change Door Open Side A';
				nFaultArrayIndex:=nFaultArrayIndex+1;
				nCurrent:=nCurrent+1;
			END_IF
		END_IF

		IF nActiveFaults[1].12=0 AND (bInCycle OR bSetup) AND NOT(bProx311) THEN
			nActiveFaults[1].12:=1;
			IF (nFaultArrayIndex<=5) THEN
				arrFaultMessage[nFaultArrayIndex]:='F013 - Tool Change Door Open Side B';
				arrFaultWarningCurrent[nCurrent]:='F013 - Tool Change Door Open Side B';
				nFaultArrayIndex:=nFaultArrayIndex+1;
				nCurrent:=nCurrent+1;
			END_IF
		END_IF

		IF nActiveFaults[1].13=0 AND (bInCycle OR bSetup) AND NOT(bProx312) THEN
			nActiveFaults[1].13:=1;
			IF (nFaultArrayIndex<=5) THEN
				arrFaultMessage[nFaultArrayIndex]:='F014 - Fixture Door Open Side A';
				arrFaultWarningCurrent[nCurrent]:='F014 - Fixture Door Open Side A';
				nFaultArrayIndex:=nFaultArrayIndex+1;
				nCurrent:=nCurrent+1;
			END_IF
		END_IF

		IF nActiveFaults[1].14=0 AND fbCycleCommonTimeout.Q THEN
			nActiveFaults[1].14:=1;
			nModeError:=Er_NoModeError;
			IF (nFaultArrayIndex<=5) THEN
				arrFaultMessage[nFaultArrayIndex]:='F015 - Cycle Start or Common Button Held Too Long';
				arrFaultWarningCurrent[nCurrent]:='F015 - Cycle Start or Common Button Held Too Long';
				nFaultArrayIndex:=nFaultArrayIndex+1;
				nCurrent:=nCurrent+1;
			END_IF
		END_IF

		IF nActiveFaults[1].15=0 AND nModeError=Er_CoolantOff THEN
			nModeError:=Er_NoModeError;
			nActiveFaults[1].15:=1;
			IF (nFaultArrayIndex<=5) THEN
				arrFaultMessage[nFaultArrayIndex]:='F016 - Coolant System Must Be On';
				arrFaultWarningCurrent[nCurrent]:='F016 - Coolant System Must Be On';
				nFaultArrayIndex:=nFaultArrayIndex+1;
				nCurrent:=nCurrent+1;
			END_IF
		END_IF

		IF nActiveFaults[1].16=0 AND nModeError=Er_VFDUpToSpeedTimeout THEN
			nModeError:=Er_NoModeError;
			nActiveFaults[1].16:=1;
			IF (nFaultArrayIndex<=5) THEN
				arrFaultMessage[nFaultArrayIndex]:='F017 - VFDs Not Up To Speed In Time';
				arrFaultWarningCurrent[nCurrent]:='F017 - VFDs Not Up To Speed In Time';
				nFaultArrayIndex:=nFaultArrayIndex+1;
				nCurrent:=nCurrent+1;
			END_IF
		END_IF

		IF nActiveFaults[1].17=0 AND nModeError=Er_AMCoolantTimeout THEN
			nActiveFaults[1].17:=1;
			nModeError:=Er_NoModeError;
			IF (nFaultArrayIndex<=5) THEN
				arrFaultMessage[nFaultArrayIndex]:='F018 - Coolant Up To Pressure Timeout';
				arrFaultWarningCurrent[nCurrent]:='F018 - Coolant Up To Pressure Timeout';
				nFaultArrayIndex:=nFaultArrayIndex+1;
				nCurrent:=nCurrent+1;
			END_IF
		END_IF

		(* If the MPG is moving the WA Axis we limit the Max Thrust for safety *)
		IF nActiveFaults[1].18=0 AND P_MPGControl.fbMPGWAAxisGearIn.InGear AND
			(ABS(nWAAxisThrust)/10 > 150)
		THEN
			bWAStop:=TRUE;	(* Stop the Axis *)
			nActiveFaults[1].18:=1;
			IF (nFaultArrayIndex<=5) THEN
				arrFaultMessage[nFaultArrayIndex]:='F019 - WA Max Thrust Exceeded';
				arrFaultWarningCurrent[nCurrent]:='F019 - WA Max Thrust Exceeded';
				nFaultArrayIndex:=nFaultArrayIndex+1;
				nCurrent:=nCurrent+1;
			END_IF
		END_IF

		(* If the MPG is moving the WA Axis limit Max Thrust to 65% for some safety *)
		IF nActiveFaults[1].19=0 AND P_MPGControl.fbMPGWBAxisGearIn.InGear AND
			ABS(nWBAxisThrust/10 > 150)
		THEN
			bWBStop:=TRUE;	(* Stop the Axis *)
			nActiveFaults[1].19:=1;
			IF (nFaultArrayIndex<=5) THEN
				arrFaultMessage[nFaultArrayIndex]:='F020 - WB Max Thrust Exceeded';
				arrFaultWarningCurrent[nCurrent]:='F020 - WB Max Thrust Exceeded';
				nFaultArrayIndex:=nFaultArrayIndex+1;
				nCurrent:=nCurrent+1;
			END_IF
		END_IF

		IF nActiveFaults[1].20=0 AND nUAxisThrust/10 > nUAxisThrustMax
			AND NOT P_MPGControl.fbMPGUAAxisGearIn.InGear
			AND NOT P_MPGControl.fbMPGXBAxisGearIn.InGear
		THEN
			nActiveFaults[1].20:=1;
			IF (nFaultArrayIndex<=5) THEN
				arrFaultMessage[nFaultArrayIndex]:='F021 - X Axis Max Thrust Exceeded';
				arrFaultWarningCurrent[nCurrent]:='F021 - X Axis Max Thrust Exceeded';
				nFaultArrayIndex:=nFaultArrayIndex+1;
				nCurrent:=nCurrent+1;
			END_IF
		END_IF

		IF nActiveFaults[1].21=0 AND nModeError=Er_TransferSolError THEN
			nModeError:=Er_NoModeError;
			nActiveFaults[1].21:=1;
			IF (nFaultArrayIndex<=5) THEN
				arrFaultMessage[nFaultArrayIndex]:='F022 - Both Up and Down Solenoids On At Same Time';
				arrFaultWarningCurrent[nCurrent]:='F022 - Both Up and Down Solenoids On At Same Time';
				nFaultArrayIndex:=nFaultArrayIndex+1;
				nCurrent:=nCurrent+1;
			END_IF
		END_IF

			IF nActiveFaults[1].22=0 AND bRack3Comm THEN
				nActiveFaults[1].22:=1;
				IF (nFaultArrayIndex<=5) THEN
					arrFaultMessage[nFaultArrayIndex]:='F023 - Com. Lost to Rack 3 Input Module';
					arrFaultWarningCurrent[nCurrent]:='F023 - Com. Lost to Rack 3 Input Module';
					nFaultArrayIndex:=nFaultArrayIndex+1;
					nCurrent:=nCurrent+1;
				END_IF
			END_IF

			IF nActiveFaults[1].23=0 AND bRack4Comm THEN
				nActiveFaults[1].23:=1;
				IF (nFaultArrayIndex<=5) THEN
					arrFaultMessage[nFaultArrayIndex]:='F024 - Com. Lost to Rack 4 Input Module';
					arrFaultWarningCurrent[nCurrent]:='F024 - Com. Lost to Rack 4 Input Module';
					nFaultArrayIndex:=nFaultArrayIndex+1;
					nCurrent:=nCurrent+1;
				END_IF
			END_IF

			IF nActiveFaults[1].24=0 AND bRack5Comm THEN
				nActiveFaults[1].24:=1;
				IF (nFaultArrayIndex<=5) THEN
					arrFaultMessage[nFaultArrayIndex]:='F025 - Com. Lost to Rack 5 Input Module';
					arrFaultWarningCurrent[nCurrent]:='F025 - Com. Lost to Rack 5 Input Module';
					nFaultArrayIndex:=nFaultArrayIndex+1;
					nCurrent:=nCurrent+1;
				END_IF
			END_IF

		IF nActiveFaults[1].25=0 AND nModeError=Er_MPG_A_Active
		THEN
			nActiveFaults[1].25:=1;
			nModeError:=Er_NoModeError;
			IF (nFaultArrayIndex<=5) THEN
				arrFaultMessage[nFaultArrayIndex]:='F026 - MPG Side A Selector Must be OFF';
				arrFaultWarningCurrent[nCurrent]:='F026 - MPG Side A Selector Must be OFF';
				nFaultArrayIndex:=nFaultArrayIndex+1;
				nCurrent:=nCurrent+1;
			END_IF
		END_IF

		IF nActiveFaults[1].26=0 AND nModeError=Er_MPG_B_Active THEN
			nActiveFaults[1].26:=1;
			nModeError:=Er_NoModeError;
			IF (nFaultArrayIndex<=5) THEN
				arrFaultMessage[nFaultArrayIndex]:='F027 - MPG Side B Selector Must be OFF';
				arrFaultWarningCurrent[nCurrent]:='F027 - MPG Side B Selector Must be OFF';
				nFaultArrayIndex:=nFaultArrayIndex+1;
				nCurrent:=nCurrent+1;
			END_IF
		END_IF

		IF nActiveFaults[1].27=0 AND bXAAxisSelected AND bXBAxisSelected THEN
			nActiveFaults[1].27:=1;
			IF (nFaultArrayIndex<=5) THEN
				arrFaultMessage[nFaultArrayIndex]:='F028 - MPG A Side and B Side Both Selected X Axis';
				arrFaultWarningCurrent[nCurrent]:='F028 - MPG A Side and B Side Both Selected X Axis';
				nFaultArrayIndex:=nFaultArrayIndex+1;
				nCurrent:=nCurrent+1;
			END_IF
		END_IF

		IF nActiveFaults[1].28=0 AND stUAxis.Status.Error  THEN
			nActiveFaults[1].28:=1;
			IF (nFaultArrayIndex<=5) THEN
				IF nUAxisDiagNumber=64720 THEN
					arrFaultMessage[nFaultArrayIndex]:='F029a - X Positive Overtravel - (+) Motion Disabled';
					arrFaultWarningCurrent[nCurrent]:='F029a - X Positive Overtravel - (+) Motion Disabled';
				ELSIF nUAxisDiagNumber=64721 THEN
					arrFaultMessage[nFaultArrayIndex]:='F029b - X Negative Overtravel - (-) Motion Disabled';
					arrFaultWarningCurrent[nCurrent]:='F029b - X Negative Overtravel - (-) Motion Disabled';
				ELSE
					arrFaultMessage[nFaultArrayIndex]:=CONCAT('F029 - Servo X Axis Fault# ',
							UDINT_TO_STRING(stUAxis.Status.ErrorID));
					arrFaultWarningCurrent[nCurrent]:=CONCAT('F029 - Servo X Axis Fault# ',
							UDINT_TO_STRING(stUAxis.Status.ErrorID));
				END_IF
				nFaultArrayIndex:=nFaultArrayIndex+1;
				nCurrent:=nCurrent+1;
			END_IF
		END_IF

		IF nActiveFaults[1].29=0 AND nModeError=Er_HomeTimeout THEN
			nActiveFaults[1].29:=1;
			nModeError:=Er_NoModeError;
			IF (nFaultArrayIndex<=5) THEN
				arrFaultMessage[nFaultArrayIndex]:='F030 - Automation Homing Did not Finish in Anticipated Time';
				arrFaultWarningCurrent[nCurrent]:='F030 - Automation Homing Did not Finish in Anticipated Time';
				nFaultArrayIndex:=nFaultArrayIndex+1;
				nCurrent:=nCurrent+1;
			END_IF
		END_IF

		IF nActiveFaults[1].30=0 AND nModeError=Er_MaxCyclesReached THEN
			nActiveFaults[1].30:=1;
			nModeError:=Er_NoModeError;
			IF (nFaultArrayIndex<=5) THEN
				arrFaultMessage[nFaultArrayIndex]:='F031 - Max Cycles Reached';
				arrFaultWarningCurrent[nCurrent]:='F031 - Max Cycles Reached';
				nFaultArrayIndex:=nFaultArrayIndex+1;
				nCurrent:=nCurrent+1;
			END_IF
		END_IF

		(***** TRANSFER FAULTS ****
		The text of the fault comes from the the TransferCycle Action of the P_TransferControl (PGM). 
			We assign the 100 series to the warnings by concating a W1 to the beginning of the text.  
			This allows us to assign the Warning series of numbers in an effort to make it more modular.  
			You must go to the function block to see the rest of the number and the description text of the fault. f
			Generally this is at the bottom of the function block or program section. 
			ErrorID < 50 is a WARNING and ErrorID >= 50 are Faults
			If this is reused in a different machine we want to make sure we assign the appropriate #series to the warnings.  *)

		IF nActiveFaults[1].31=0 AND bTransferError  AND nTransferErrorID >= 50THEN
			nActiveFaults[1].31:=1;
			IF (nFaultArrayIndex<=5) THEN
				arrFaultMessage[nFaultArrayIndex]:=CONCAT('F1',sTransferErrorText);
				arrFaultWarningCurrent[nCurrent]:=CONCAT('F1',sTransferErrorText);
				nFaultArrayIndex:=nFaultArrayIndex+1;
				nCurrent:=nCurrent+1;
			END_IF
		END_IF

	(* 	SIDE A FAULTS
		The text of the fault comes from the function block "Side_A_Fixture" and we assign the hundreds series # to it below.
		Example: Side A Fixture has F2 is concated to the front of the text so that they are 200 series faults
				Side B fixture has F3 concated to make them 300 series faults..  
		You must go to the function block to see the rest of the number and the description text of the fault. 
		Generally this is at the bottom of the function block. *)
		IF bSideAEnabled THEN
			(* Tailstock Side A *)
			IF nActiveFaults[2].0=0 AND Side_A_Fixture.bError THEN
				nActiveFaults[2].0:=1;
				IF (nFaultArrayIndex<=5) THEN
					arrFaultMessage[nFaultArrayIndex]:=CONCAT('F2',Side_A_Fixture.sErrorText);
						arrFaultMessage[nFaultArrayIndex]:=CONCAT(arrFaultMessage[nFaultArrayIndex],' Side A');
					arrFaultWarningCurrent[nCurrent]:=CONCAT('F2',Side_A_Fixture.sErrorText);
						arrFaultWarningCurrent[nCurrent]:=CONCAT(arrFaultWarningCurrent[nCurrent],' Side A');
					nFaultArrayIndex:=nFaultArrayIndex+1;
					nCurrent:=nCurrent+1;
				END_IF
			END_IF

			IF nActiveFaults[2].1=0 AND bACoolantSolenoid
				AND bLowFlow1A AND NOT(fCoolantFlowMin<0.5)
				AND fbFlowAverageTimer1ALOW.Q AND fbCoolantOnDelayTON.Q
			THEN
				nActiveFaults[2].1:=1;
				IF (nFaultArrayIndex<=5) THEN
					arrFaultMessage[nFaultArrayIndex]:='F230 - Coolant Flow Below Min #1A';
					arrFaultWarningCurrent[nCurrent]:='F230 - Coolant Flow Below Min #1A';
					nFaultArrayIndex:=nFaultArrayIndex+1;
					nCurrent:=nCurrent+1;
				END_IF
			END_IF

			IF nActiveFaults[2].2=0 AND bACoolantSolenoid
				AND bHighFlow1A AND NOT(fCoolantFlowMax=60)
				AND fbFlowAverageTimer1AHIGH.Q AND fbCoolantOnDelayTON.Q
			THEN
				nActiveFaults[2].2:=1;
				IF (nFaultArrayIndex<=5) THEN
					arrFaultMessage[nFaultArrayIndex]:='F231 - Coolant Flow Exceeded Max #1A';
					arrFaultWarningCurrent[nCurrent]:='F231 - Coolant Flow Exceeded Max #1A';
					nFaultArrayIndex:=nFaultArrayIndex+1;
					nCurrent:=nCurrent+1;
				END_IF
			END_IF

			IF nActiveFaults[2].3=0 AND bACoolantSolenoid
				AND bLowFlow2A AND NOT(fCoolantFlowMin<0.5)
				AND fbFlowAverageTimer2ALOW.Q AND fbCoolantOnDelayTON.Q
			THEN
				nActiveFaults[2].3:=1;
				IF (nFaultArrayIndex<=5) THEN
					arrFaultMessage[nFaultArrayIndex]:='F232 - Coolant Flow Below Min #2A';
					arrFaultWarningCurrent[nCurrent]:='F232 - Coolant Flow Below Min #2A';
					nFaultArrayIndex:=nFaultArrayIndex+1;
					nCurrent:=nCurrent+1;
				END_IF
			END_IF

			IF nActiveFaults[2].4=0 AND bACoolantSolenoid
				AND bHighFlow2A AND NOT(fCoolantFlowMax=60)
				AND fbFlowAverageTimer2AHIGH.Q AND fbCoolantOnDelayTON.Q
			THEN
				nActiveFaults[2].4:=1;
				IF (nFaultArrayIndex<=5) THEN
					arrFaultMessage[nFaultArrayIndex]:='F233 - Coolant Flow Exceeded Max #2A';
					arrFaultWarningCurrent[nCurrent]:='F233 - Coolant Flow Exceeded Max #2A';
					nFaultArrayIndex:=nFaultArrayIndex+1;
					nCurrent:=nCurrent+1;
				END_IF
			END_IF

			IF nActiveFaults[2].5=0 AND bACoolantSolenoid
				AND bLowFlow3A AND NOT(fCoolantFlowMin<0.5)
				AND fbFlowAverageTimer3ALOW.Q AND fbCoolantOnDelayTON.Q
			THEN
				nActiveFaults[2].5:=1;
				IF (nFaultArrayIndex<=5) THEN
					arrFaultMessage[nFaultArrayIndex]:='F234 - Coolant Flow Below Min #3A';
					arrFaultWarningCurrent[nCurrent]:='F234 - Coolant Flow Below Min #3A';
					nFaultArrayIndex:=nFaultArrayIndex+1;
					nCurrent:=nCurrent+1;
				END_IF
			END_IF
			IF nActiveFaults[2].6=0 AND bACoolantSolenoid
				AND bHighFlow3A AND NOT(fCoolantFlowMax=60)
				AND fbFlowAverageTimer3AHIGH.Q AND fbCoolantOnDelayTON.Q
			THEN
				nActiveFaults[2].6:=1;
				IF (nFaultArrayIndex<=5) THEN
					arrFaultMessage[nFaultArrayIndex]:='F235 - Coolant Flow Exceeded Max #3A';
					arrFaultWarningCurrent[nCurrent]:='F235 - Coolant Flow Exceeded Max #3A';
					nFaultArrayIndex:=nFaultArrayIndex+1;
					nCurrent:=nCurrent+1;
				END_IF
			END_IF

			IF nActiveFaults[2].7=0 AND NOT(nServoThrustMax=0) AND fbServoAThrustMaxDelayTON.Q
				AND bInCycle AND NOT(stZAAxis.Status.InPositionArea) AND (stZAAxis.NcToPlc.AxisState=3) THEN
				nActiveFaults[2].7:=1;
				IF (nFaultArrayIndex<=5) THEN
					arrFaultMessage[nFaultArrayIndex]:='F236 - Servo ZA Thrust Exceeded Max';
					arrFaultWarningCurrent[nCurrent]:='F236 - Servo  ZAThrust Exceeded Max';
					nFaultArrayIndex:=nFaultArrayIndex+1;
					nCurrent:=nCurrent+1;
				END_IF
			END_IF

			IF nActiveFaults[2].8=0 AND stZAAxis.Status.Error  THEN
				nActiveFaults[2].8:=1;
				IF (nFaultArrayIndex<=5) THEN
 					IF nZAAxisDiagNumber=64720 THEN
						arrFaultMessage[nFaultArrayIndex]:='F237a - ZA Negative Overtravel - (-) Motion Disabled';
						arrFaultWarningCurrent[nCurrent]:='F237a - ZA Negative Overtravel - (-) Motion Disabled';
					ELSIF nZAAxisDiagNumber=64721 THEN
						arrFaultMessage[nFaultArrayIndex]:='F237b - ZA  Positive Overtravel - (+) Motion Disabled';
						arrFaultWarningCurrent[nCurrent]:='F237b - ZA Positive Overtravel - (+) Motion Disabled';
					ELSE
						arrFaultMessage[nFaultArrayIndex]:=CONCAT('F237 - Servo ZA Axis Fault# ',
								UDINT_TO_STRING(stZAAxis.Status.ErrorID));
						arrFaultWarningCurrent[nCurrent]:=CONCAT('F237 - Servo ZA Axis Fault# ',
								UDINT_TO_STRING(stZAAxis.Status.ErrorID));
					END_IF
					nFaultArrayIndex:=nFaultArrayIndex+1;
					nCurrent:=nCurrent+1;
				END_IF
			END_IF

			IF nActiveFaults[2].9=0 AND stWAAxis.Status.Error  THEN
				nActiveFaults[2].9:=1;
				IF (nFaultArrayIndex<=5) THEN
 					IF nWAAxisDiagNumber=64720 THEN
						arrFaultMessage[nFaultArrayIndex]:='F238a - WA Negative Overtravel - (-) Motion Disabled';
						arrFaultWarningCurrent[nCurrent]:='F238a - WA Negative Overtravel - (-) Motion Disabled';
					ELSIF nWAAxisDiagNumber=64721 THEN
						arrFaultMessage[nFaultArrayIndex]:='F238b - WA  Positive Overtravel - (+) Motion Disabled';
						arrFaultWarningCurrent[nCurrent]:='F238b - WA  Positive Overtravel - (+) Motion Disabled';
					ELSE
						arrFaultMessage[nFaultArrayIndex]:=CONCAT('F238 - Servo WA Axis Fault# ',
							UDINT_TO_STRING(stWAAxis.Status.ErrorID));
						arrFaultWarningCurrent[nCurrent]:=CONCAT('F238 - Servo WA Axis Fault# ',
							UDINT_TO_STRING(stWAAxis.Status.ErrorID));
					END_IF
					nFaultArrayIndex:=nFaultArrayIndex+1;
					nCurrent:=nCurrent+1;
				END_IF
			END_IF

			IF nActiveFaults[2].10=0 AND fbWAAxisHome.Error  THEN
				nActiveFaults[2].10:=1;
				IF (nFaultArrayIndex<=5) THEN
					arrFaultMessage[nFaultArrayIndex]:='F239 - Tailstock WA Homing Error';
					arrFaultWarningCurrent[nCurrent]:='F239 - Tailstock WA Homing Error';;
					nFaultArrayIndex:=nFaultArrayIndex+1;
					nCurrent:=nCurrent+1;
				END_IF
			END_IF

			IF nActiveFaults[2].11=0 AND nSpindleLoad1ADisplay>nSpindleLoadMax AND NOT(nSpindleLoadMax=0)
				AND bVFD_ARun AND bVFD_A1UpToSpeed AND fbALoadFaultDelay.Q THEN
				 nActiveFaults[2].11:=1;
				IF (nFaultArrayIndex<=5) THEN
					arrFaultMessage[nFaultArrayIndex]:='F240 - Spindle #1A Max Load Exceeded';
					arrFaultWarningCurrent[nCurrent]:='F240 - Spindle #1A Max Load Exceeded';
					nFaultArrayIndex:=nFaultArrayIndex+1;
					nCurrent:=nCurrent+1;
				END_IF
			END_IF
	
			IF nActiveFaults[2].12=0 AND nSpindleLoad2ADisplay>nSpindleLoadMax AND NOT(nSpindleLoadMax=0)
				AND bVFD_ARun AND bVFD_A2UpToSpeed AND fbALoadFaultDelay.Q THEN
				 nActiveFaults[2].12:=1;
				IF (nFaultArrayIndex<=5) THEN
					arrFaultMessage[nFaultArrayIndex]:='F241 - Spindle #2A Max Load Exceeded';
					arrFaultWarningCurrent[nCurrent]:='F241 - Spindle #2A Max Load Exceeded';
					nFaultArrayIndex:=nFaultArrayIndex+1;
					nCurrent:=nCurrent+1;
				END_IF
			END_IF

			IF nActiveFaults[2].13=0 AND nSpindleLoad3ADisplay>nSpindleLoadMax AND NOT(nSpindleLoadMax=0)
				AND bVFD_ARun AND bVFD_A3UpToSpeed AND fbALoadFaultDelay.Q THEN
				 nActiveFaults[2].13:=1;
				IF (nFaultArrayIndex<=5) THEN
					arrFaultMessage[nFaultArrayIndex]:='F242 - Spindle #3A Max Load Exceeded';
					arrFaultWarningCurrent[nCurrent]:='F242 - Spindle #3A Max Load Exceeded';
					nFaultArrayIndex:=nFaultArrayIndex+1;
					nCurrent:=nCurrent+1;
				END_IF
			END_IF

		(* Spares - Future Spindles *)

			IF nActiveFaults[2].18=0 AND fbVFD_A1.bError THEN
			(*	Encompasses ALL VFD related Errors *)
			(* uptospeed, drivenotready, drivefaulted, drivewarning, drivecomm *)
				nActiveFaults[2].18:=1;
				IF (nFaultArrayIndex<=5) THEN
					IF fbVFD_A1.nErrorID=Er_DriveComm THEN
						arrFaultMessage[nFaultArrayIndex]:='F243a - Spindle #1A VFD Communcation Failed';
						arrFaultWarningCurrent[nCurrent]:='F243a - Spindle #1A VFD Communcation Failed';
						nFaultArrayIndex:=nFaultArrayIndex+1;
						nCurrent:=nCurrent+1;
					ELSIF fbVFD_A1.nErrorID=Er_DriveFaulted THEN
						arrFaultMessage[nFaultArrayIndex]:='F243b - Spindle #1A VFD Fault';
						arrFaultWarningCurrent[nCurrent]:='F243b - Spindle #1A VFD Fault';
						nFaultArrayIndex:=nFaultArrayIndex+1;
						nCurrent:=nCurrent+1;
					ELSIF fbVFD_A1.nErrorID=Er_DriveWarning THEN
						arrFaultMessage[nFaultArrayIndex]:='F243c - Spindle #1A VFD Warning';
						arrFaultWarningCurrent[nCurrent]:='F243c - Spindle #1A VFD Warning';
						nFaultArrayIndex:=nFaultArrayIndex+1;
						nCurrent:=nCurrent+1;
					ELSIF fbVFD_A1.nErrorID=Er_DriveNotReady THEN
						arrFaultMessage[nFaultArrayIndex]:='F243d - Spindle #1A VFD Not Ready';
						arrFaultWarningCurrent[nCurrent]:='F243d - Spindle #1A VFD Not Ready';
						nFaultArrayIndex:=nFaultArrayIndex+1;
						nCurrent:=nCurrent+1;
					ELSIF fbVFD_A1.nErrorID=Er_InvalidRPM THEN
						arrFaultMessage[nFaultArrayIndex]:='F243e - Spindle #1A VFD Invalid RPM Requested';
						arrFaultWarningCurrent[nCurrent]:='F243e - Spindle #1A VFD Invalid RPM Requested';
						nFaultArrayIndex:=nFaultArrayIndex+1;
						nCurrent:=nCurrent+1;
					ELSIF fbVFD_A1.nErrorID=Er_InvalidRatio THEN
						arrFaultMessage[nFaultArrayIndex]:='F243f - Spindle #1A VFD Invalid Motor to Spindle Ratio Requested';
						arrFaultWarningCurrent[nCurrent]:='F243f - Spindle #1A VFD Invalid Motor to Spindle Ratio Requested';
						nFaultArrayIndex:=nFaultArrayIndex+1;
						nCurrent:=nCurrent+1;
					ELSIF fbVFD_A1.nErrorID=Er_InvalidOverride THEN
						arrFaultMessage[nFaultArrayIndex]:='F243g - Spindle #1A VFD Invalid Override Requested';
						arrFaultWarningCurrent[nCurrent]:='F243g - Spindle #1A VFD Invalid Override Requested';
						nFaultArrayIndex:=nFaultArrayIndex+1;
						nCurrent:=nCurrent+1;
					ELSIF fbVFD_A1.nErrorID=Er_UpToSpeedTimeout THEN
						arrFaultMessage[nFaultArrayIndex]:='F243h - Spindle #1A VFD Not Up To Speed';
						arrFaultWarningCurrent[nCurrent]:='F243h - Spindle #1A VFD Not Up To Speed';
						nFaultArrayIndex:=nFaultArrayIndex+1;
						nCurrent:=nCurrent+1;
					ELSE
						arrFaultMessage[nFaultArrayIndex]:=CONCAT('F243 - Spindle #1A VFD Error : ',
												UDINT_TO_STRING(fbVFD_A1.stVFDInfo.nActiveFault));
						arrFaultWarningCurrent[nCurrent]:=CONCAT('F243 - Spindle #1A VFD Error : ',
												UDINT_TO_STRING(fbVFD_A1.stVFDInfo.nActiveFault));
						nFaultArrayIndex:=nFaultArrayIndex+1;
						nCurrent:=nCurrent+1;
					END_IF
				END_IF
			END_IF

			IF nActiveFaults[2].19=0 AND fbVFD_A2.bError THEN
			(*	Encompasses ALL VFD related Errors *)
			(* uptospeed, drivenotready, drivefaulted, drivewarning, drivecomm *)
				nActiveFaults[2].19:=1;
				IF (nFaultArrayIndex<=5) THEN
					IF fbVFD_A2.nErrorID=Er_DriveComm THEN
						arrFaultMessage[nFaultArrayIndex]:='F244a - Spindle #2A VFD Communcation Failed';
						arrFaultWarningCurrent[nCurrent]:='F244a - Spindle #2A VFD Communcation Failed';
						nFaultArrayIndex:=nFaultArrayIndex+1;
						nCurrent:=nCurrent+1;
					ELSIF fbVFD_A2.nErrorID=Er_DriveFaulted THEN
						arrFaultMessage[nFaultArrayIndex]:='F244b - Spindle #2A VFD Fault';
						arrFaultWarningCurrent[nCurrent]:='F244b - Spindle #2A VFD Fault';
						nFaultArrayIndex:=nFaultArrayIndex+1;
						nCurrent:=nCurrent+1;
					ELSIF fbVFD_A2.nErrorID=Er_DriveWarning THEN
						arrFaultMessage[nFaultArrayIndex]:='F244c - Spindle #2A VFD Warning';
						arrFaultWarningCurrent[nCurrent]:='F244c - Spindle #2A VFD Warning';
						nFaultArrayIndex:=nFaultArrayIndex+1;
						nCurrent:=nCurrent+1;
					ELSIF fbVFD_A2.nErrorID=Er_DriveNotReady THEN
						arrFaultMessage[nFaultArrayIndex]:='F244d - Spindle #2A VFD Not Ready';
						arrFaultWarningCurrent[nCurrent]:='F244d - Spindle #2A VFD Not Ready';
						nFaultArrayIndex:=nFaultArrayIndex+1;
						nCurrent:=nCurrent+1;
					ELSIF fbVFD_A2.nErrorID=Er_InvalidRPM THEN
						arrFaultMessage[nFaultArrayIndex]:='F244e - Spindle #2A VFD Invalid RPM Requested';
						arrFaultWarningCurrent[nCurrent]:='F244e - Spindle #2A VFD Invalid RPM Requested';
						nFaultArrayIndex:=nFaultArrayIndex+1;
						nCurrent:=nCurrent+1;
					ELSIF fbVFD_A2.nErrorID=Er_InvalidRatio THEN
						arrFaultMessage[nFaultArrayIndex]:='F244f - Spindle #2A VFD Invalid Motor to Spindle Ratio Requested';
						arrFaultWarningCurrent[nCurrent]:='F244f - Spindle #2A VFD Invalid Motor to Spindle Ratio Requested';
						nFaultArrayIndex:=nFaultArrayIndex+1;
						nCurrent:=nCurrent+1;
					ELSIF fbVFD_A2.nErrorID=Er_InvalidOverride THEN
						arrFaultMessage[nFaultArrayIndex]:='F244g - Spindle #2A VFD Invalid Override Requested';
						arrFaultWarningCurrent[nCurrent]:='F244g - Spindle #2A VFD Invalid Override Requested';
						nFaultArrayIndex:=nFaultArrayIndex+1;
						nCurrent:=nCurrent+1;
					ELSIF fbVFD_A2.nErrorID=Er_UpToSpeedTimeout THEN
						arrFaultMessage[nFaultArrayIndex]:='F244h - Spindle #2A VFD Not Up To Speed';
						arrFaultWarningCurrent[nCurrent]:='F244h - Spindle #2A VFD Not Up To Speed';
						nFaultArrayIndex:=nFaultArrayIndex+1;
						nCurrent:=nCurrent+1;
					ELSE
						arrFaultMessage[nFaultArrayIndex]:=CONCAT('F244 - Spindle #2A VFD Error : ',
												UDINT_TO_STRING(fbVFD_A2.stVFDInfo.nActiveFault));
						arrFaultWarningCurrent[nCurrent]:=CONCAT('F244 - Spindle #2A VFD Error : ',
												UDINT_TO_STRING(fbVFD_A2.stVFDInfo.nActiveFault));
						nFaultArrayIndex:=nFaultArrayIndex+1;
						nCurrent:=nCurrent+1;
					END_IF
				END_IF
			END_IF

			IF nActiveFaults[2].20=0 AND fbVFD_A3.bError THEN
			(*	Encompasses ALL VFD related Errors *)
			(* uptospeed, drivenotready, drivefaulted, drivewarning, drivecomm *)
				nActiveFaults[2].20:=1;
				IF (nFaultArrayIndex<=5) THEN
					IF fbVFD_A3.nErrorID=Er_DriveComm THEN
						arrFaultMessage[nFaultArrayIndex]:='F245a - Spindle #3A VFD Communcation Failed';
						arrFaultWarningCurrent[nCurrent]:='F245a - Spindle #3A VFD Communcation Failed';
						nFaultArrayIndex:=nFaultArrayIndex+1;
						nCurrent:=nCurrent+1;
					ELSIF fbVFD_A3.nErrorID=Er_DriveFaulted THEN
						arrFaultMessage[nFaultArrayIndex]:='F245b - Spindle #3A VFD Fault';
						arrFaultWarningCurrent[nCurrent]:='F245b - Spindle #3A VFD Fault';
						nFaultArrayIndex:=nFaultArrayIndex+1;
						nCurrent:=nCurrent+1;
					ELSIF fbVFD_A3.nErrorID=Er_DriveWarning THEN
						arrFaultMessage[nFaultArrayIndex]:='F245c - Spindle #3A VFD Warning';
						arrFaultWarningCurrent[nCurrent]:='F245c - Spindle #3A VFD Warning';
						nFaultArrayIndex:=nFaultArrayIndex+1;
						nCurrent:=nCurrent+1;
					ELSIF fbVFD_A3.nErrorID=Er_DriveNotReady THEN
						arrFaultMessage[nFaultArrayIndex]:='F245d - Spindle #3A VFD Not Ready';
						arrFaultWarningCurrent[nCurrent]:='F245d - Spindle #3A VFD Not Ready';
						nFaultArrayIndex:=nFaultArrayIndex+1;
						nCurrent:=nCurrent+1;
					ELSIF fbVFD_A3.nErrorID=Er_InvalidRPM THEN
						arrFaultMessage[nFaultArrayIndex]:='F245e - Spindle #3A VFD Invalid RPM Requested';
						arrFaultWarningCurrent[nCurrent]:='F245e - Spindle #3A VFD Invalid RPM Requested';
						nFaultArrayIndex:=nFaultArrayIndex+1;
						nCurrent:=nCurrent+1;
					ELSIF fbVFD_A3.nErrorID=Er_InvalidRatio THEN
						arrFaultMessage[nFaultArrayIndex]:='F245f - Spindle #3A VFD Invalid Motor to Spindle Ratio Requested';
						arrFaultWarningCurrent[nCurrent]:='F245f - Spindle #3A VFD Invalid Motor to Spindle Ratio Requested';
						nFaultArrayIndex:=nFaultArrayIndex+1;
						nCurrent:=nCurrent+1;
					ELSIF fbVFD_A3.nErrorID=Er_InvalidOverride THEN
						arrFaultMessage[nFaultArrayIndex]:='F245g - Spindle #3A VFD Invalid Override Requested';
						arrFaultWarningCurrent[nCurrent]:='F245g - Spindle #3A VFD Invalid Override Requested';
						nFaultArrayIndex:=nFaultArrayIndex+1;
						nCurrent:=nCurrent+1;
					ELSIF fbVFD_A3.nErrorID=Er_UpToSpeedTimeout THEN
						arrFaultMessage[nFaultArrayIndex]:='F245h - Spindle #3A VFD Not Up To Speed';
						arrFaultWarningCurrent[nCurrent]:='F245h - Spindle #3A VFD Not Up To Speed';
						nFaultArrayIndex:=nFaultArrayIndex+1;
						nCurrent:=nCurrent+1;
					ELSE
						arrFaultMessage[nFaultArrayIndex]:=CONCAT('F245 - Spindle #3A VFD Error : ',
												UDINT_TO_STRING(fbVFD_A3.stVFDInfo.nActiveFault));
						arrFaultWarningCurrent[nCurrent]:=CONCAT('F245 - Spindle #3A VFD Error : ',
												UDINT_TO_STRING(fbVFD_A3.stVFDInfo.nActiveFault));
						nFaultArrayIndex:=nFaultArrayIndex+1;
						nCurrent:=nCurrent+1;
					END_IF
				END_IF
			END_IF

			(* Coolant Pressure Fault for Auto Mode *)
			IF nActiveFaults[2].21=0 AND fbLowPressureFaultADelay.Q
				AND bMachineMode
			THEN
				nActiveFaults[2].21:=1;
				IF (nFaultArrayIndex<=5) THEN
					arrFaultMessage[nFaultArrayIndex]:='F246 - Coolant Pressure Low - Side A';
					arrFaultWarningCurrent[nCurrent]:='F246 - Coolant Pressure Low - Side A';
					nFaultArrayIndex:=nFaultArrayIndex+1;
					nCurrent:=nCurrent+1;
				END_IF
			END_IF

			IF nActiveFaults[2].22=0 AND fbSpeedVariationTimer1AHIGH.Q
				AND bVFD_ARun  AND bVFD_A1UpToSpeed AND (bInCycle OR bSetupA)
				AND fbASpeedDelayTimer.Q THEN
				nActiveFaults[2].22:=1;
				IF (nFaultArrayIndex<=5) THEN
					arrFaultMessage[nFaultArrayIndex]:='F247 - Spindle Speed Not Correct #1A (HIGH)';
					arrFaultWarningCurrent[nCurrent]:='F247 - Spindle Speed Not Correct #1A (HIGH)';
					nFaultArrayIndex:=nFaultArrayIndex+1;
					nCurrent:=nCurrent+1;
				END_IF
			END_IF

			IF nActiveFaults[2].23=0 AND fbSpeedVariationTimer1ALOW.Q
				AND bVFD_ARun AND bVFD_A1UpToSpeed AND (bInCycle OR bSetupA)
				AND fbASpeedDelayTimer.Q THEN
				nActiveFaults[2].23:=1;
				IF (nFaultArrayIndex<=5) THEN
					arrFaultMessage[nFaultArrayIndex]:='F248 - Spindle Speed Not Correct #1A (LOW)';
					arrFaultWarningCurrent[nCurrent]:='F248 - Spindle Speed Not Correct #1A (LOW)';
					nFaultArrayIndex:=nFaultArrayIndex+1;
					nCurrent:=nCurrent+1;
				END_IF
			END_IF
	
			IF nActiveFaults[2].24=0 AND fbSpeedVariationTimer2AHIGH.Q
				AND bVFD_ARun  AND bVFD_A2UpToSpeed AND (bInCycle OR bSetupA)
				AND fbASpeedDelayTimer.Q THEN
				nActiveFaults[2].24:=1;
				IF (nFaultArrayIndex<=5) THEN
					arrFaultMessage[nFaultArrayIndex]:='F249 - Spindle Speed Not Correct #2A (HIGH)';
					arrFaultWarningCurrent[nCurrent]:='F249 - Spindle Speed Not Correct #2A (HIGH)';
					nFaultArrayIndex:=nFaultArrayIndex+1;
					nCurrent:=nCurrent+1;
				END_IF
			END_IF
			IF nActiveFaults[2].25=0 AND fbSpeedVariationTimer2ALOW.Q
				AND bVFD_ARun AND bVFD_A2UpToSpeed AND (bInCycle OR bSetupA)
				AND fbASpeedDelayTimer.Q THEN
				nActiveFaults[2].25:=1;
				IF (nFaultArrayIndex<=5) THEN
					arrFaultMessage[nFaultArrayIndex]:='F250 - Spindle Speed Not Correct #2A (LOW)';
					arrFaultWarningCurrent[nCurrent]:='F250- Spindle Speed Not Correct #2A (LOW)';
					nFaultArrayIndex:=nFaultArrayIndex+1;
					nCurrent:=nCurrent+1;
				END_IF
			END_IF
	
			IF nActiveFaults[2].26=0 AND fbSpeedVariationTimer3AHIGH.Q
				AND bVFD_ARun  AND bVFD_A3UpToSpeed AND (bInCycle OR bSetupA)
				AND fbASpeedDelayTimer.Q THEN
				nActiveFaults[2].26:=1;
				IF (nFaultArrayIndex<=5) THEN
					arrFaultMessage[nFaultArrayIndex]:='F251 - Spindle Speed Not Correct #3A (HIGH)';
					arrFaultWarningCurrent[nCurrent]:='F251 - Spindle Speed Not Correct #3A (HIGH)';
					nFaultArrayIndex:=nFaultArrayIndex+1;
					nCurrent:=nCurrent+1;
				END_IF
			END_IF

			IF nActiveFaults[2].27=0 AND fbSpeedVariationTimer3ALOW.Q
				AND bVFD_ARun AND bVFD_A3UpToSpeed AND (bInCycle OR bSetupA)
				AND fbASpeedDelayTimer.Q THEN
				nActiveFaults[2].27:=1;
				IF (nFaultArrayIndex<=5) THEN
					arrFaultMessage[nFaultArrayIndex]:='F252 - Spindle Speed Not Correct #3A (LOW)';
					arrFaultWarningCurrent[nCurrent]:='F252 - Spindle Speed Not Correct #3A (LOW)';
					nFaultArrayIndex:=nFaultArrayIndex+1;
					nCurrent:=nCurrent+1;
				END_IF
			END_IF

			IF nActiveFaults[2].28=0 AND nModeError=Er_SideAColletSolError THEN
				nModeError:=Er_NoModeError;
				nActiveFaults[2].28:=1;
				IF (nFaultArrayIndex<=5) THEN
					arrFaultMessage[nFaultArrayIndex]:='F253 - Both A Clamp and UnClamp Solenoids On At Same Time';
					arrFaultWarningCurrent[nCurrent]:='F253 - Both A Clamp and UnClamp Solenoids On At Same Time';
					nFaultArrayIndex:=nFaultArrayIndex+1;
					nCurrent:=nCurrent+1;
				END_IF
			END_IF

			IF nActiveFaults[2].29=0 AND nModeError=Er_SideAEjectorsSolError THEN
				nModeError:=Er_NoModeError;
				nActiveFaults[2].29:=1;
				IF (nFaultArrayIndex<=5) THEN
					arrFaultMessage[nFaultArrayIndex]:='F254 - Both A Ejector Advance  and Retract Solenoids On At Same Time';
					arrFaultWarningCurrent[nCurrent]:='F254 - Both A Ejector Advance  and Retract Solenoids On At Same Time';
					nFaultArrayIndex:=nFaultArrayIndex+1;
					nCurrent:=nCurrent+1;
				END_IF
			END_IF

			IF nActiveFaults[2].30=0 AND bRack6Comm THEN
				nActiveFaults[2].30:=1;
				IF (nFaultArrayIndex<=5) THEN
					arrFaultMessage[nFaultArrayIndex]:='F255 - Com. Lost to Side A Tailstock Input Module';
					arrFaultWarningCurrent[nCurrent]:='F255 - Com. Lost to Side A Tailstock Input Module';;
					nFaultArrayIndex:=nFaultArrayIndex+1;
					nCurrent:=nCurrent+1;
				END_IF
			END_IF

